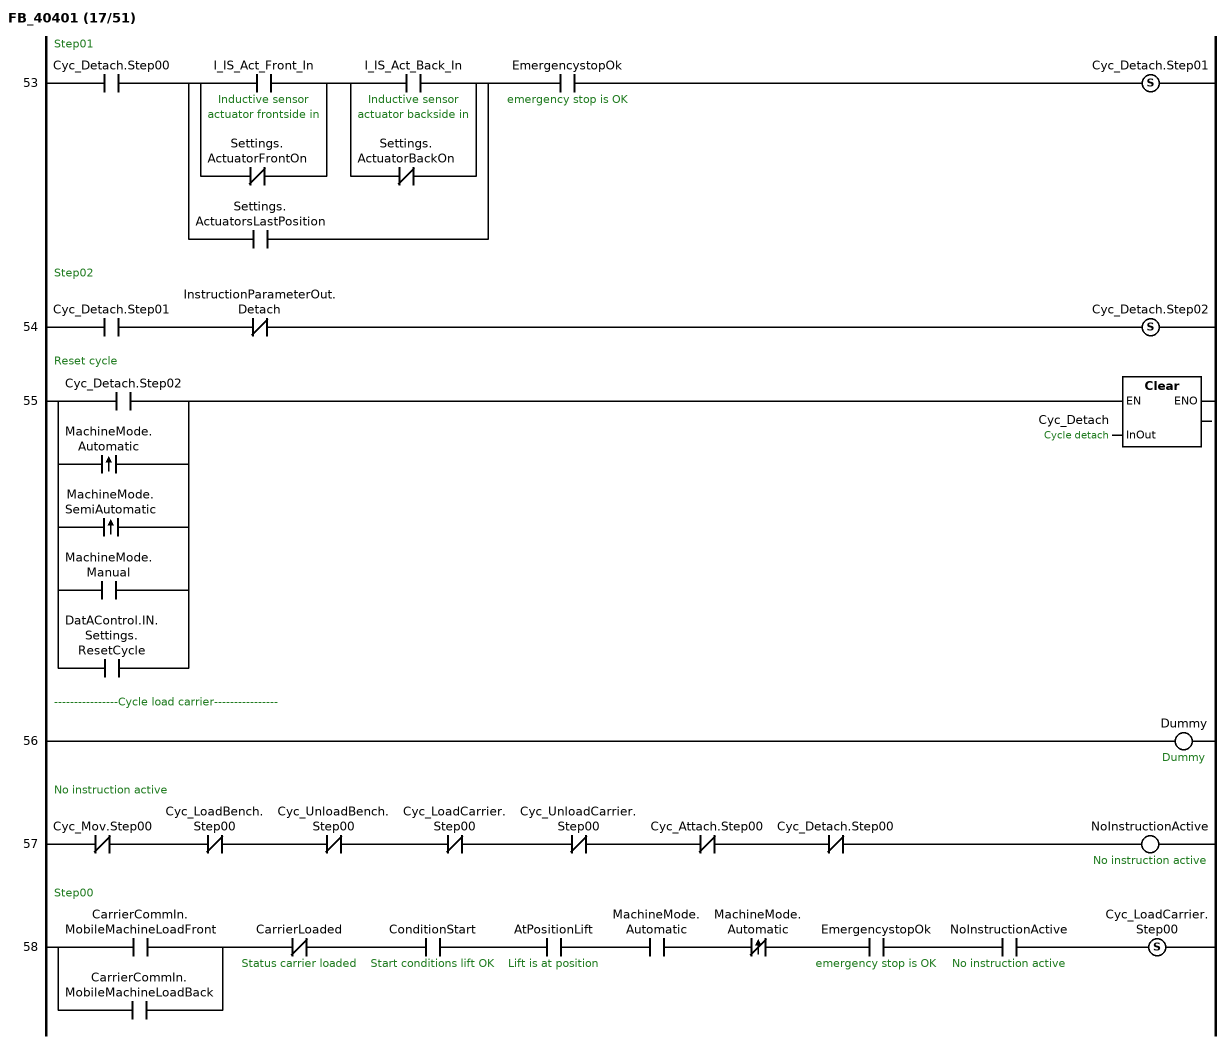
(* [picture p150: FB_40401, rungs 53-58] *)
(* Rung 53: Step01 *)
IF Cyc_Detach.Step00 AND (((I_IS_Act_Front_In OR NOT Settings.ActuatorFrontOn) AND (I_IS_Act_Back_In OR NOT Settings.ActuatorBackOn)) OR Settings.ActuatorsLastPosition) AND EmergencystopOk THEN
    Cyc_Detach.Step01 := TRUE;
END_IF;
(* Rung 54: Step02 *)
IF Cyc_Detach.Step01 AND NOT InstructionParameterOut.Detach THEN Cyc_Detach.Step02 := TRUE; END_IF;
(* Rung 55: Reset cycle *)
_e31(CLK := MachineMode.Automatic);
_e32(CLK := MachineMode.SemiAutomatic);
IF Cyc_Detach.Step02 OR _e31.Q OR _e32.Q OR MachineMode.Manual OR DatAControl.IN.Settings.ResetCycle THEN
    Clear(InOut := Cyc_Detach);
END_IF;
(* Rung 56: ----------------Cycle load carrier---------------- *)
Dummy := TRUE;
(* Rung 57: No instruction active *)
NoInstructionActive := NOT Cyc_Mov.Step00 AND NOT Cyc_LoadBench.Step00 AND NOT Cyc_UnloadBench.Step00 AND NOT Cyc_LoadCarrier.Step00 AND NOT Cyc_UnloadCarrier.Step00 AND NOT Cyc_Attach.Step00 AND NOT Cyc_Detach.Step00;
(* Rung 58: Step00 *)
_e33(CLK := MachineMode.Automatic);
IF (CarrierCommIn.MobileMachineLoadFront OR CarrierCommIn.MobileMachineLoadBack) AND NOT CarrierLoaded AND ConditionStart AND AtPositionLift AND MachineMode.Automatic AND NOT _e33.Q AND EmergencystopOk AND NoInstructionActive THEN
    Cyc_LoadCarrier.Step00 := TRUE;
END_IF;

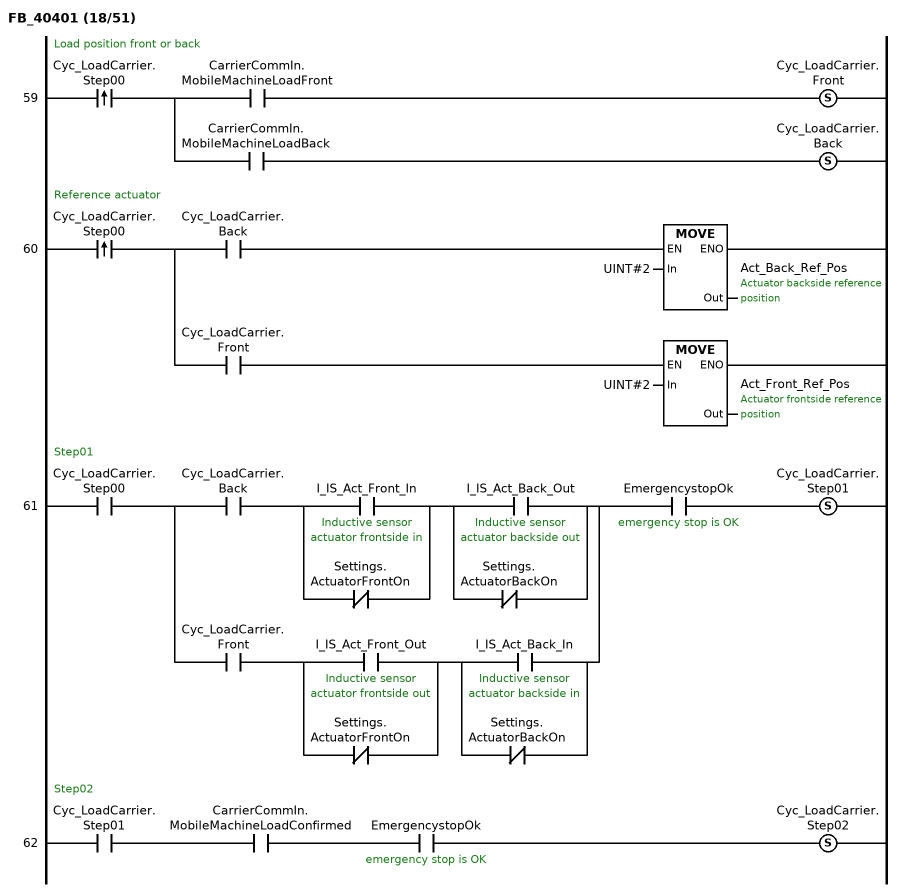
(* Rung 59: Load position front or back *)
_e34(CLK := Cyc_LoadCarrier.Step00);
IF _e34.Q AND CarrierCommIn.MobileMachineLoadFront THEN Cyc_LoadCarrier.Front := TRUE; END_IF;
IF _e34.Q AND CarrierCommIn.MobileMachineLoadBack THEN Cyc_LoadCarrier.Back := TRUE; END_IF;
(* Rung 60: Reference actuator *)
_e35(CLK := Cyc_LoadCarrier.Step00);
IF _e35.Q AND Cyc_LoadCarrier.Back THEN Act_Back_Ref_Pos := UINT#2; END_IF;
IF _e35.Q AND Cyc_LoadCarrier.Front THEN Act_Front_Ref_Pos := UINT#2; END_IF;
(* Rung 61: Step01 *)
IF Cyc_LoadCarrier.Step00 AND ((Cyc_LoadCarrier.Back AND (I_IS_Act_Front_In OR NOT Settings.ActuatorFrontOn) AND (I_IS_Act_Back_Out OR NOT Settings.ActuatorBackOn)) OR (Cyc_LoadCarrier.Front AND (I_IS_Act_Front_Out OR NOT Settings.ActuatorFrontOn) AND (I_IS_Act_Back_In OR NOT Settings.ActuatorBackOn))) AND EmergencystopOk THEN
    Cyc_LoadCarrier.Step01 := TRUE;
END_IF;
(* Rung 62: Step02 *)
IF Cyc_LoadCarrier.Step01 AND CarrierCommIn.MobileMachineLoadConfirmed AND EmergencystopOk THEN
    Cyc_LoadCarrier.Step02 := TRUE;
END_IF;

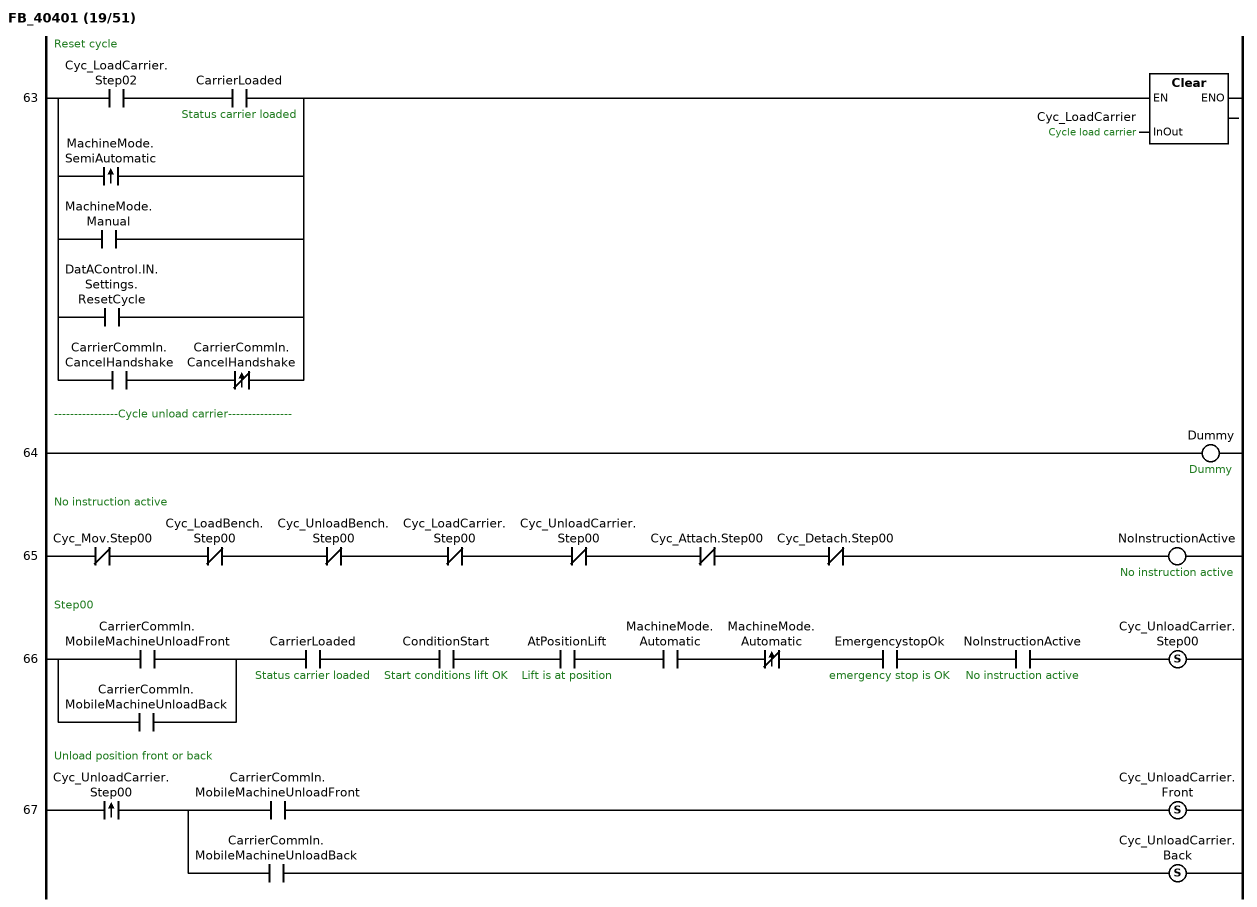
(* Rung 63: Reset cycle *)
_e36(CLK := MachineMode.SemiAutomatic);
_e37(CLK := CarrierCommIn.CancelHandshake);
IF (Cyc_LoadCarrier.Step02 AND CarrierLoaded) OR _e36.Q OR MachineMode.Manual OR DatAControl.IN.Settings.ResetCycle OR (CarrierCommIn.CancelHandshake AND NOT _e37.Q) THEN
    Clear(InOut := Cyc_LoadCarrier);
END_IF;
(* Rung 64: ----------------Cycle unload carrier---------------- *)
Dummy := TRUE;
(* Rung 65: No instruction active *)
NoInstructionActive := NOT Cyc_Mov.Step00 AND NOT Cyc_LoadBench.Step00 AND NOT Cyc_UnloadBench.Step00 AND NOT Cyc_LoadCarrier.Step00 AND NOT Cyc_UnloadCarrier.Step00 AND NOT Cyc_Attach.Step00 AND NOT Cyc_Detach.Step00;
(* Rung 66: Step00 *)
_e38(CLK := MachineMode.Automatic);
IF (CarrierCommIn.MobileMachineUnloadFront OR CarrierCommIn.MobileMachineUnloadBack) AND CarrierLoaded AND ConditionStart AND AtPositionLift AND MachineMode.Automatic AND NOT _e38.Q AND EmergencystopOk AND NoInstructionActive THEN
    Cyc_UnloadCarrier.Step00 := TRUE;
END_IF;
(* Rung 67: Unload position front or back *)
_e39(CLK := Cyc_UnloadCarrier.Step00);
IF _e39.Q AND CarrierCommIn.MobileMachineUnloadFront THEN Cyc_UnloadCarrier.Front := TRUE; END_IF;
IF _e39.Q AND CarrierCommIn.MobileMachineUnloadBack THEN Cyc_UnloadCarrier.Back := TRUE; END_IF;

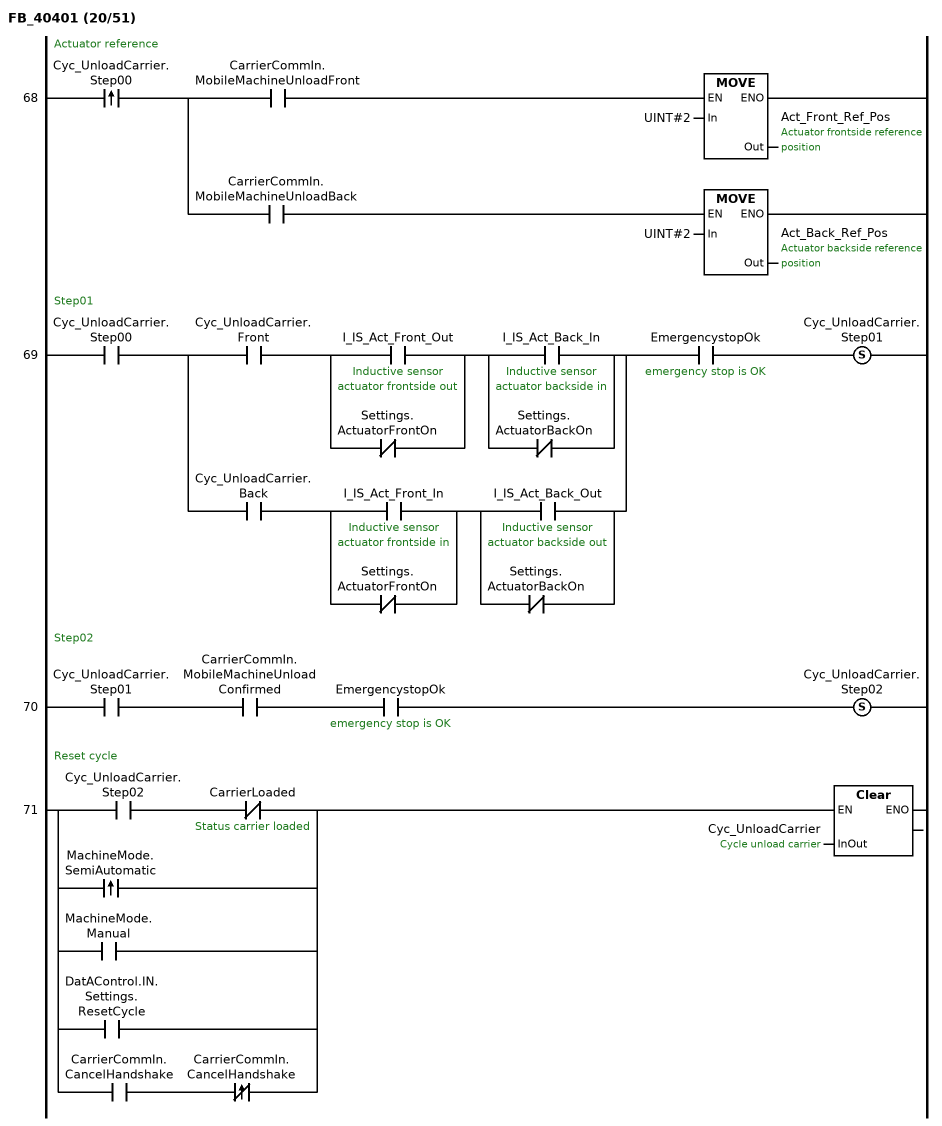
(* Rung 68: Actuator reference *)
_e40(CLK := Cyc_UnloadCarrier.Step00);
IF _e40.Q AND CarrierCommIn.MobileMachineUnloadFront THEN Act_Front_Ref_Pos := UINT#2; END_IF;
IF _e40.Q AND CarrierCommIn.MobileMachineUnloadBack THEN Act_Back_Ref_Pos := UINT#2; END_IF;
(* Rung 69: Step01 *)
IF Cyc_UnloadCarrier.Step00 AND ((Cyc_UnloadCarrier.Front AND (I_IS_Act_Front_Out OR NOT Settings.ActuatorFrontOn) AND (I_IS_Act_Back_In OR NOT Settings.ActuatorBackOn)) OR (Cyc_UnloadCarrier.Back AND (I_IS_Act_Front_In OR NOT Settings.ActuatorFrontOn) AND (I_IS_Act_Back_Out OR NOT Settings.ActuatorBackOn))) AND EmergencystopOk THEN
    Cyc_UnloadCarrier.Step01 := TRUE;
END_IF;
(* Rung 70: Step02 *)
IF Cyc_UnloadCarrier.Step01 AND CarrierCommIn.MobileMachineUnloadConfirmed AND EmergencystopOk THEN
    Cyc_UnloadCarrier.Step02 := TRUE;
END_IF;
(* Rung 71: Reset cycle *)
_e41(CLK := MachineMode.SemiAutomatic);
_e42(CLK := CarrierCommIn.CancelHandshake);
IF (Cyc_UnloadCarrier.Step02 AND NOT CarrierLoaded) OR _e41.Q OR MachineMode.Manual OR DatAControl.IN.Settings.ResetCycle OR (CarrierCommIn.CancelHandshake AND NOT _e42.Q) THEN
    Clear(InOut := Cyc_UnloadCarrier);
END_IF;

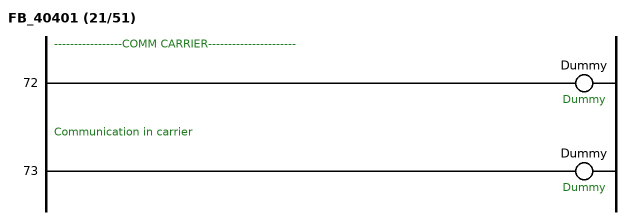
(* Rung 72: -----------------COMM CARRIER---------------------- *)
Dummy := TRUE;
(* Rung 73: Communication in carrier *)
Dummy := TRUE;

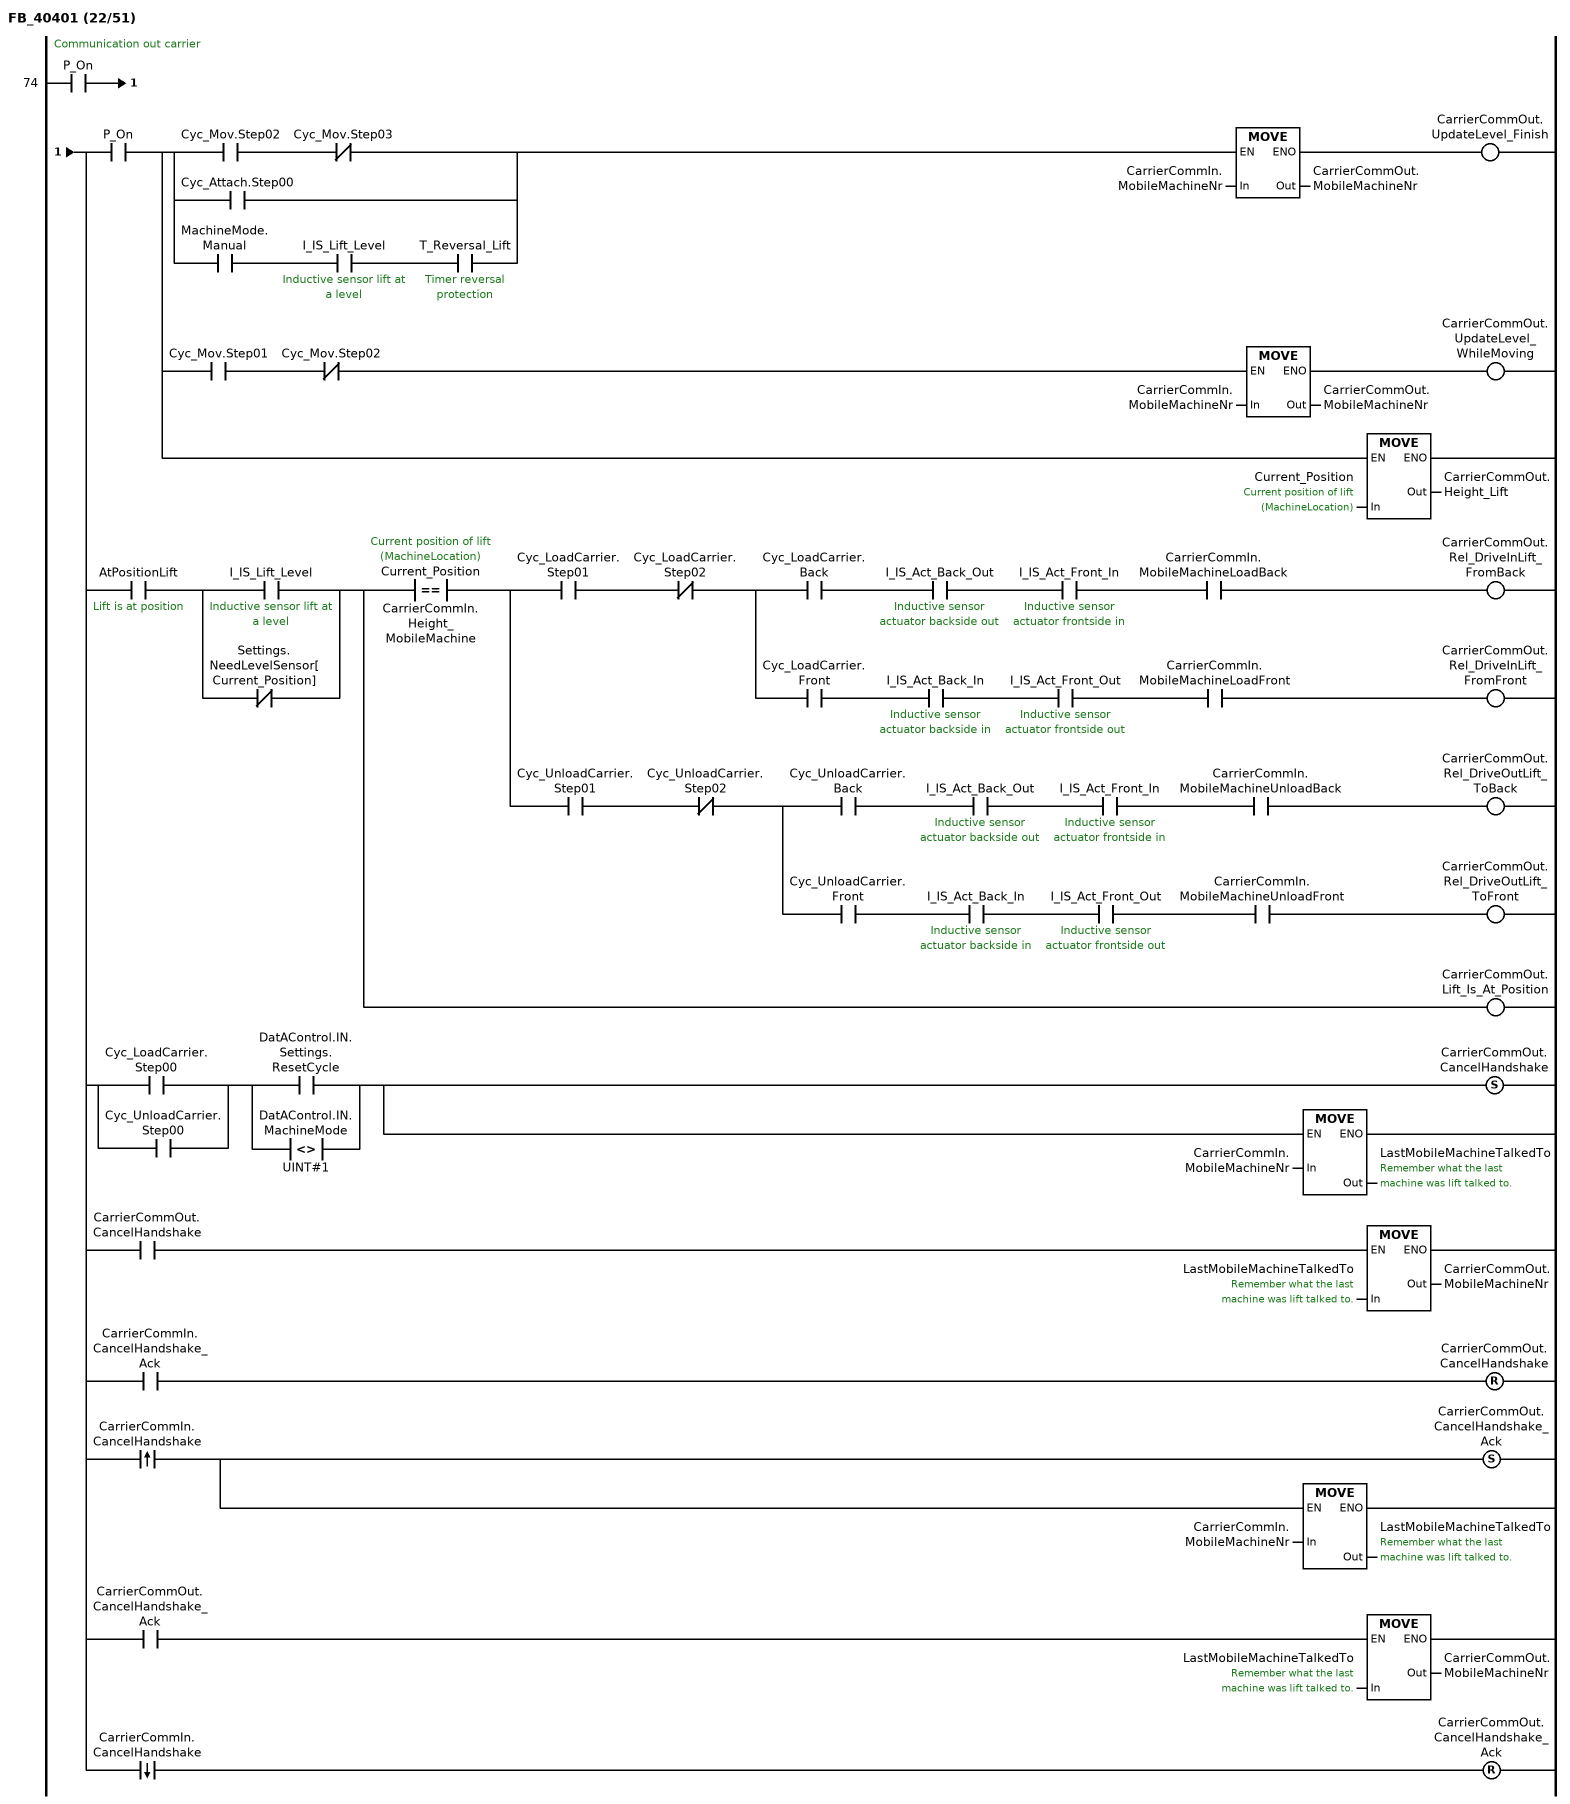
(* Rung 74: Communication out carrier *)
IF P_On AND P_On AND ((Cyc_Mov.Step02 AND NOT Cyc_Mov.Step03) OR Cyc_Attach.Step00 OR (MachineMode.Manual AND I_IS_Lift_Level AND T_Reversal_Lift)) THEN
    CarrierCommOut.MobileMachineNr := CarrierCommIn.MobileMachineNr;
END_IF;
CarrierCommOut.UpdateLevel_Finish := P_On AND P_On AND ((Cyc_Mov.Step02 AND NOT Cyc_Mov.Step03) OR Cyc_Attach.Step00 OR (MachineMode.Manual AND I_IS_Lift_Level AND T_Reversal_Lift));
IF P_On AND P_On AND Cyc_Mov.Step01 AND NOT Cyc_Mov.Step02 THEN
    CarrierCommOut.MobileMachineNr := CarrierCommIn.MobileMachineNr;
END_IF;
CarrierCommOut.UpdateLevel_WhileMoving := P_On AND P_On AND Cyc_Mov.Step01 AND NOT Cyc_Mov.Step02;
IF P_On AND P_On THEN CarrierCommOut.Height_Lift := Current_Position; END_IF;
_p43 := P_On AND AtPositionLift AND (I_IS_Lift_Level OR NOT Settings.NeedLevelSensor[Current_Position]);
_p44 := _p43 AND (Current_Position = CarrierCommIn.Height_MobileMachine);
_p45 := _p44 AND Cyc_LoadCarrier.Step01 AND NOT Cyc_LoadCarrier.Step02;
CarrierCommOut.Rel_DriveInLift_FromBack := _p45 AND Cyc_LoadCarrier.Back AND I_IS_Act_Back_Out AND I_IS_Act_Front_In AND CarrierCommIn.MobileMachineLoadBack;
CarrierCommOut.Rel_DriveInLift_FromFront := _p45 AND Cyc_LoadCarrier.Front AND I_IS_Act_Back_In AND I_IS_Act_Front_Out AND CarrierCommIn.MobileMachineLoadFront;
_p46 := _p44 AND Cyc_UnloadCarrier.Step01 AND NOT Cyc_UnloadCarrier.Step02;
CarrierCommOut.Rel_DriveOutLift_ToBack := _p46 AND Cyc_UnloadCarrier.Back AND I_IS_Act_Back_Out AND I_IS_Act_Front_In AND CarrierCommIn.MobileMachineUnloadBack;
CarrierCommOut.Rel_DriveOutLift_ToFront := _p46 AND Cyc_UnloadCarrier.Front AND I_IS_Act_Back_In AND I_IS_Act_Front_Out AND CarrierCommIn.MobileMachineUnloadFront;
CarrierCommOut.Lift_Is_At_Position := _p43;
_p47 := P_On AND (Cyc_LoadCarrier.Step00 OR Cyc_UnloadCarrier.Step00) AND (DatAControl.IN.Settings.ResetCycle OR (DatAControl.IN.MachineMode <> UINT#1));
IF _p47 THEN
    CarrierCommOut.CancelHandshake := TRUE;
    LastMobileMachineTalkedTo := CarrierCommIn.MobileMachineNr;
END_IF;
IF P_On AND CarrierCommOut.CancelHandshake THEN
    CarrierCommOut.MobileMachineNr := LastMobileMachineTalkedTo;
END_IF;
IF P_On AND CarrierCommIn.CancelHandshake_Ack THEN CarrierCommOut.CancelHandshake := FALSE; END_IF;
_e48(CLK := CarrierCommIn.CancelHandshake);
IF P_On AND _e48.Q THEN
    CarrierCommOut.CancelHandshake_Ack := TRUE;
    LastMobileMachineTalkedTo := CarrierCommIn.MobileMachineNr;
END_IF;
IF P_On AND CarrierCommOut.CancelHandshake_Ack THEN
    CarrierCommOut.MobileMachineNr := LastMobileMachineTalkedTo;
END_IF;
_e49(CLK := CarrierCommIn.CancelHandshake);
IF P_On AND _e49.Q THEN CarrierCommOut.CancelHandshake_Ack := FALSE; END_IF;

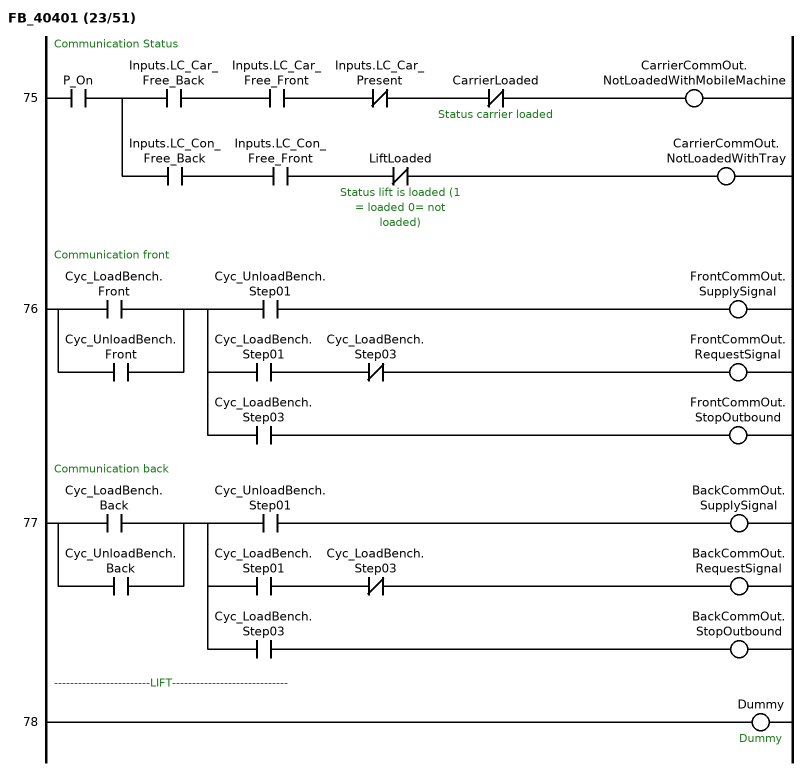
(* Rung 75: Communication Status *)
CarrierCommOut.NotLoadedWithMobileMachine := P_On AND Inputs.LC_Car_Free_Back AND Inputs.LC_Car_Free_Front AND NOT Inputs.LC_Car_Present AND NOT CarrierLoaded;
CarrierCommOut.NotLoadedWithTray := P_On AND Inputs.LC_Con_Free_Back AND Inputs.LC_Con_Free_Front AND NOT LiftLoaded;
(* Rung 76: Communication front *)
FrontCommOut.SupplySignal := (Cyc_LoadBench.Front OR Cyc_UnloadBench.Front) AND Cyc_UnloadBench.Step01;
FrontCommOut.RequestSignal := (Cyc_LoadBench.Front OR Cyc_UnloadBench.Front) AND Cyc_LoadBench.Step01 AND NOT Cyc_LoadBench.Step03;
FrontCommOut.StopOutbound := (Cyc_LoadBench.Front OR Cyc_UnloadBench.Front) AND Cyc_LoadBench.Step03;
(* Rung 77: Communication back *)
BackCommOut.SupplySignal := (Cyc_LoadBench.Back OR Cyc_UnloadBench.Back) AND Cyc_UnloadBench.Step01;
BackCommOut.RequestSignal := (Cyc_LoadBench.Back OR Cyc_UnloadBench.Back) AND Cyc_LoadBench.Step01 AND NOT Cyc_LoadBench.Step03;
BackCommOut.StopOutbound := (Cyc_LoadBench.Back OR Cyc_UnloadBench.Back) AND Cyc_LoadBench.Step03;
(* Rung 78: ------------------------LIFT----------------------------- *)
Dummy := TRUE;

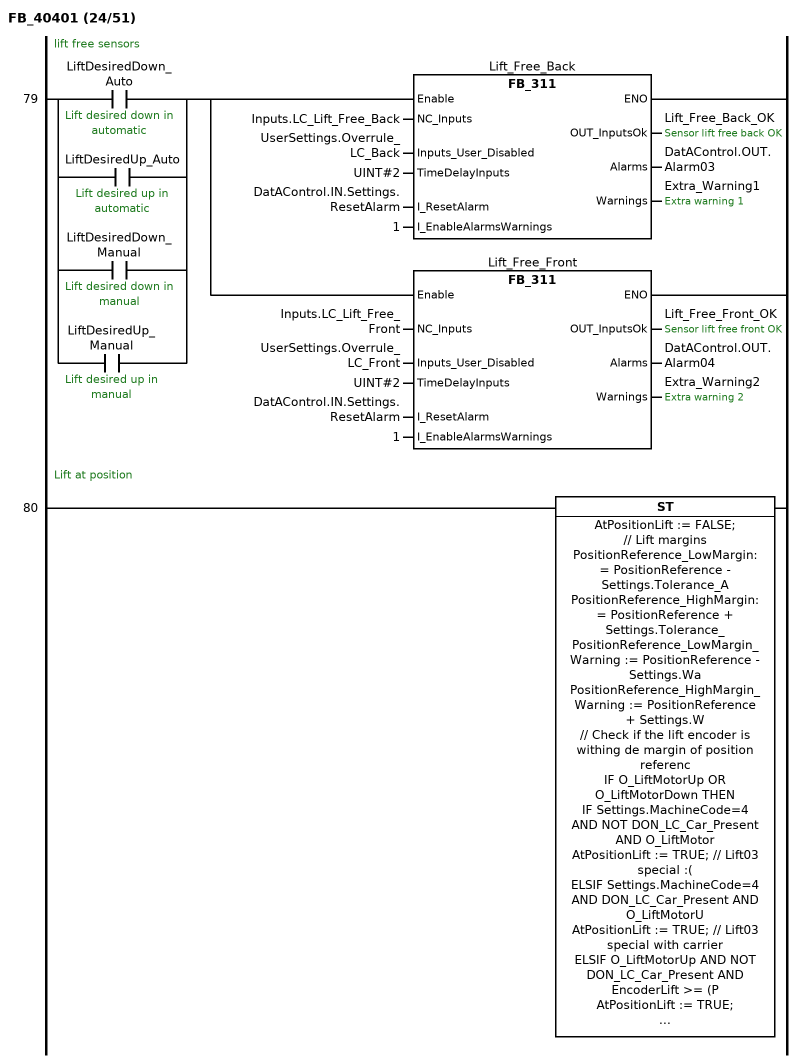
(* Rung 79: lift free sensors *)
_p50 := LiftDesiredDown_Auto OR LiftDesiredUp_Auto OR LiftDesiredDown_Manual OR LiftDesiredUp_Manual;
Lift_Free_Back(Enable := _p50, NC_Inputs := Inputs.LC_Lift_Free_Back, Inputs_User_Disabled := UserSettings.Overrule_LC_Back, TimeDelayInputs := UINT#2, I_ResetAlarm := DatAControl.IN.Settings.ResetAlarm, I_EnableAlarmsWarnings := 1, OUT_InputsOk => Lift_Free_Back_OK, Alarms => DatAControl.OUT.Alarm03, Warnings => Extra_Warning1);
Lift_Free_Front(Enable := _p50, NC_Inputs := Inputs.LC_Lift_Free_Front, Inputs_User_Disabled := UserSettings.Overrule_LC_Front, TimeDelayInputs := UINT#2, I_ResetAlarm := DatAControl.IN.Settings.ResetAlarm, I_EnableAlarmsWarnings := 1, OUT_InputsOk => Lift_Free_Front_OK, Alarms => DatAControl.OUT.Alarm04, Warnings => Extra_Warning2);
(* Rung 80: Lift at position *)
AtPositionLift := FALSE;

// Lift margins
PositionReference_LowMargin:= PositionReference - Settings.Tolerance_At_Position;
PositionReference_HighMargin:= PositionReference + Settings.Tolerance_At_Position;
PositionReference_LowMargin_Warning := PositionReference - Settings.Warning_Tolerance_At_Position;
PositionReference_HighMargin_Warning := PositionReference + Settings.Warning_Tolerance_At_Position;

// Check if the lift encoder is withing de margin of position reference
IF O_LiftMotorUp OR O_LiftMotorDown THEN
	IF Settings.MachineCode=4 AND NOT DON_LC_Car_Present AND O_LiftMotorUp AND EncoderLift >= (PositionReference + 25) AND EncoderLift <= (PositionReference_HighMargin) THEN // EncoderLiftOvershootUp
		AtPositionLift := TRUE; // Lift03 special :(
	ELSIF Settings.MachineCode=4 AND DON_LC_Car_Present AND O_LiftMotorUp AND EncoderLift >= (PositionReference + 25) AND EncoderLift <= (PositionReference_HighMargin) THEN
		AtPositionLift := TRUE; // Lift03 special with carrier
	ELSIF O_LiftMotorUp AND NOT DON_LC_Car_Present AND EncoderLift >= (PositionReference - EncoderLiftOvershootUp) AND EncoderLift <= PositionReference_HighMargin THEN
		AtPositionLift := TRUE;
	ELSIF O_LiftMotorUp AND DON_LC_Car_Present AND EncoderLift >= (PositionReference - EncoderLiftOvershootUp - EncoderLiftOvershootUp) AND EncoderLift <= PositionReference_HighMargin THEN
		AtPositionLift := TRUE; // with carrier
	ELSIF Settings.MachineCode=4 AND O_LiftMotorDown AND NOT DON_LC_Car_Present AND EncoderLift <= (PositionReference + 45) AND EncoderLift >= PositionReference_LowMargin  THEN
		AtPositionLift := TRUE; // Lift03 special :)
	ELSIF Settings.MachineCode=4 AND O_LiftMotorDown AND DON_LC_Car_Present AND EncoderLift <= (PositionReference + 45) AND EncoderLift >= PositionReference_LowMargin  THEN
		AtPositionLift := TRUE; // Lift03 special with carrier
	ELSIF O_LiftMotorDown AND NOT DON_LC_Car_Present AND EncoderLift <= (PositionReference + EncoderLiftOvershootDown) AND EncoderLift >= PositionReference_LowMargin THEN
		AtPositionLift := TRUE;
	ELSIF O_LiftMotorDown AND DON_LC_Car_Present AND EncoderLift <= (PositionReference + EncoderLiftOvershootDown + EncoderLiftOvershootDown) AND EncoderLift >= PositionReference_LowMargin THEN
		AtPositionLift := TRUE; // with carrier
	END_IF;
ELSE
	IF (EncoderLift >= PositionReference_LowMargin) AND (EncoderLift <= PositionReference_HighMargin) THEN
		AtPositionLift := TRUE;
	END_IF;
END_IF;

Warning_AtPositionLift := FALSE;
IF AtPositionLift AND T_Reversal_Lift AND ((EncoderLift <= PositionReference_LowMargin_Warning) OR (EncoderLift >= PositionReference_HighMargin_Warning)) THEN
	Warning_AtPositionLift := TRUE;
END_IF;

Extra_Warning3 := WORD#0;

IF Warning_AtPositionLift THEN
	OutABit(Extra_Warning3,0,TRUE);
END_IF;

// Check for each position if the lift encoder is within the margins
FOR index:=1 TO 16 BY 1 DO
	IF (EncoderLift >= ( Settings.PulseLevel[index] - Settings.Tolerance_At_Position)) AND (EncoderLift <= (Settings.PulseLevel[index] + Settings.Tolerance_At_Position)) THEN
		Current_Position:= index;
	END_IF;
END_FOR;

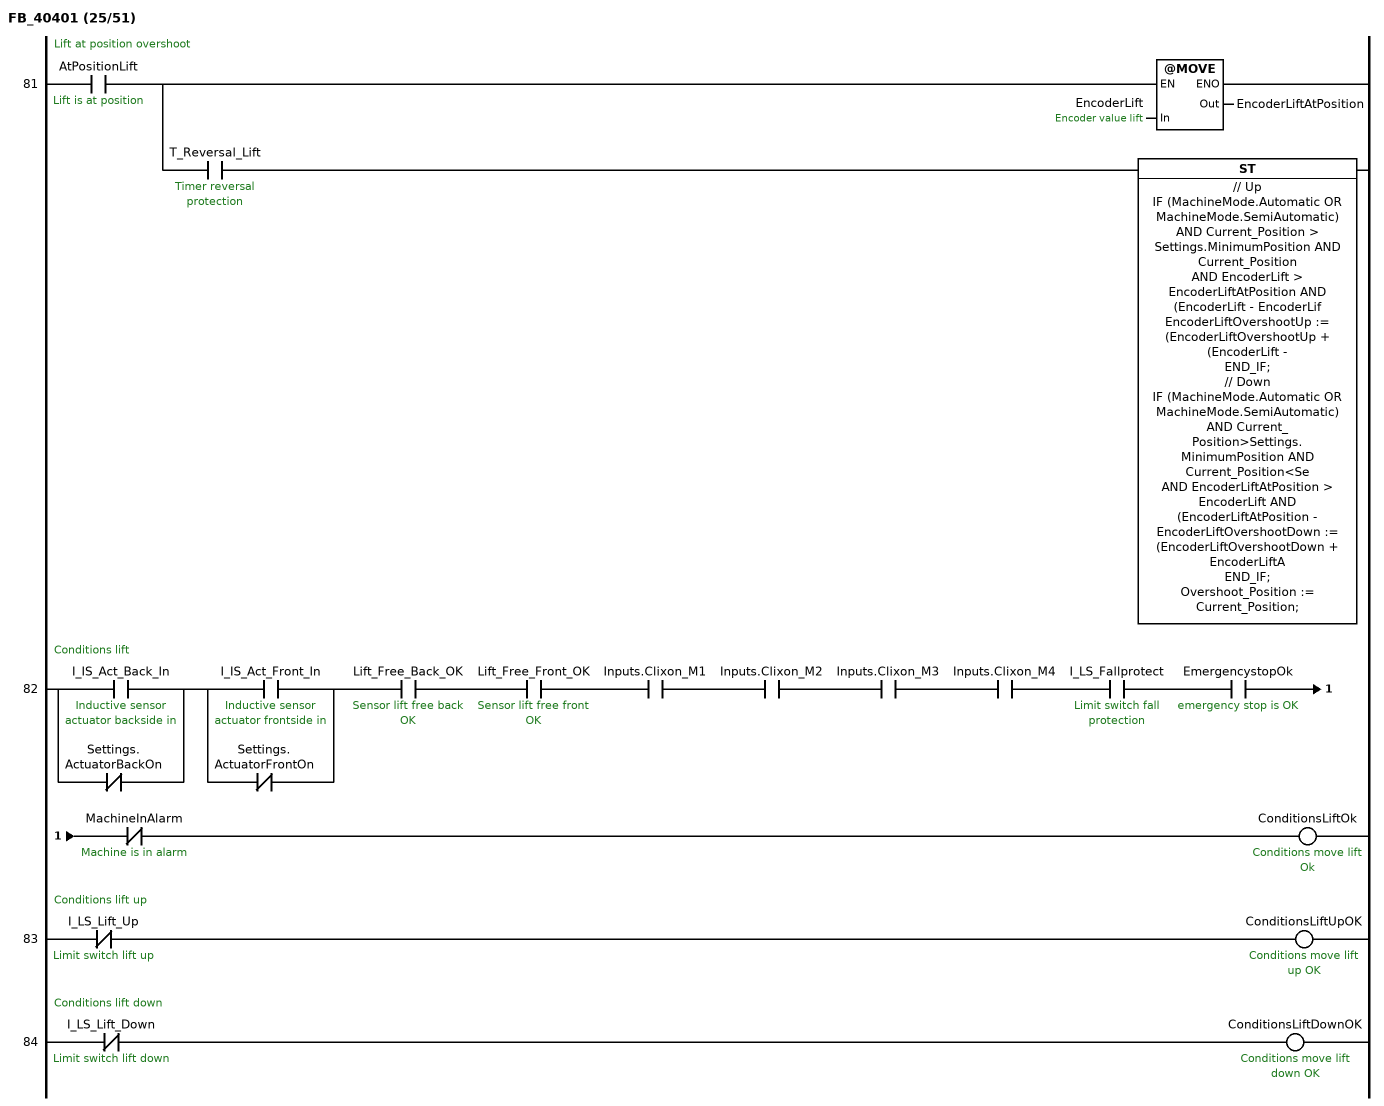
(* Rung 81: Lift at position overshoot *)
_e51(CLK := AtPositionLift);
IF _e51.Q THEN EncoderLiftAtPosition := EncoderLift; END_IF;
IF AtPositionLift AND T_Reversal_Lift THEN
    // Up
    IF (MachineMode.Automatic OR MachineMode.SemiAutomatic)
     AND Current_Position > Settings.MinimumPosition AND Current_Position < Settings.MaximumPosition AND Current_Position <> Overshoot_Position
     AND EncoderLift > EncoderLiftAtPosition AND (EncoderLift - EncoderLiftAtPosition) < (Settings.Tolerance_At_Position*2) THEN
    		EncoderLiftOvershootUp := (EncoderLiftOvershootUp + (EncoderLift - EncoderLiftAtPosition))/2;
    END_IF;
    // Down
    IF (MachineMode.Automatic OR MachineMode.SemiAutomatic)
     AND Current_Position>Settings.MinimumPosition AND Current_Position<Settings.MaximumPosition AND Current_Position<>Overshoot_Position
     AND EncoderLiftAtPosition > EncoderLift AND (EncoderLiftAtPosition - EncoderLift) < (Settings.Tolerance_At_Position*2) THEN
    	EncoderLiftOvershootDown := (EncoderLiftOvershootDown + EncoderLiftAtPosition - EncoderLift)/2;
    END_IF;
    
    Overshoot_Position := Current_Position;
END_IF;
(* Rung 82: Conditions lift *)
ConditionsLiftOk := (I_IS_Act_Back_In OR NOT Settings.ActuatorBackOn) AND (I_IS_Act_Front_In OR NOT Settings.ActuatorFrontOn) AND Lift_Free_Back_OK AND Lift_Free_Front_OK AND Inputs.Clixon_M1 AND Inputs.Clixon_M2 AND Inputs.Clixon_M3 AND Inputs.Clixon_M4 AND I_LS_Fallprotect AND EmergencystopOk AND NOT MachineInAlarm;
(* Rung 83: Conditions lift up *)
ConditionsLiftUpOK := NOT I_LS_Lift_Up;
(* Rung 84: Conditions lift down *)
ConditionsLiftDownOK := NOT I_LS_Lift_Down;

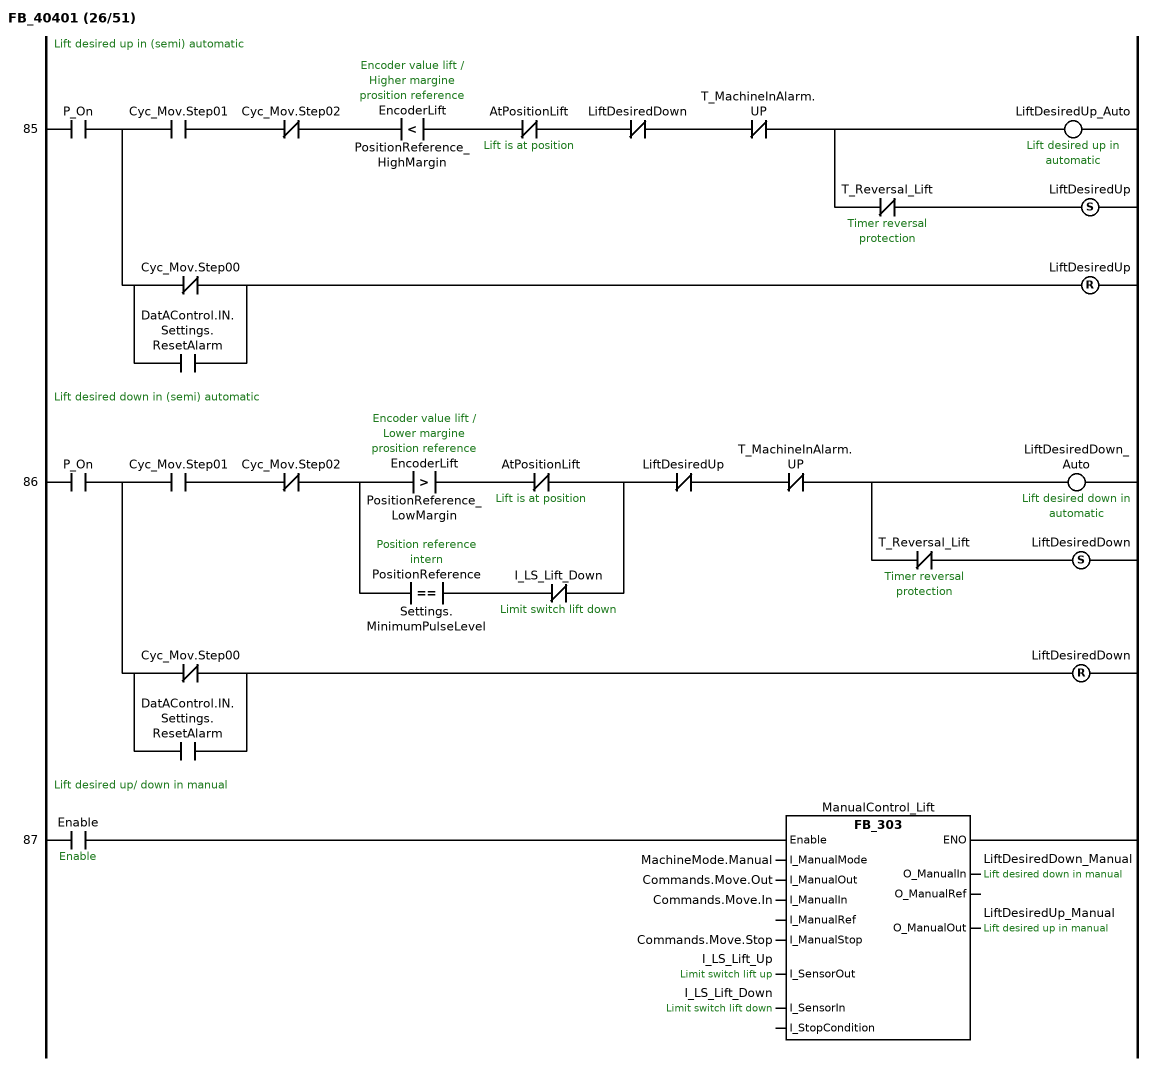
(* Rung 85: Lift desired up in (semi) automatic *)
_p52 := P_On AND Cyc_Mov.Step01 AND NOT Cyc_Mov.Step02 AND (EncoderLift < PositionReference_HighMargin) AND NOT AtPositionLift AND NOT LiftDesiredDown AND NOT T_MachineInAlarm.UP;
LiftDesiredUp_Auto := _p52;
IF _p52 AND NOT T_Reversal_Lift THEN LiftDesiredUp := TRUE; END_IF;
IF P_On AND (NOT Cyc_Mov.Step00 OR DatAControl.IN.Settings.ResetAlarm) THEN
    LiftDesiredUp := FALSE;
END_IF;
(* Rung 86: Lift desired down in (semi) automatic *)
_p53 := P_On AND Cyc_Mov.Step01 AND NOT Cyc_Mov.Step02 AND (((EncoderLift > PositionReference_LowMargin) AND NOT AtPositionLift) OR ((PositionReference = Settings.MinimumPulseLevel) AND NOT I_LS_Lift_Down)) AND NOT LiftDesiredUp AND NOT T_MachineInAlarm.UP;
LiftDesiredDown_Auto := _p53;
IF _p53 AND NOT T_Reversal_Lift THEN LiftDesiredDown := TRUE; END_IF;
IF P_On AND (NOT Cyc_Mov.Step00 OR DatAControl.IN.Settings.ResetAlarm) THEN
    LiftDesiredDown := FALSE;
END_IF;
(* Rung 87: Lift desired up/ down in manual *)
ManualControl_Lift(Enable := Enable, I_ManualMode := MachineMode.Manual, I_ManualOut := Commands.Move.Out, I_ManualIn := Commands.Move.In, I_ManualStop := Commands.Move.Stop, I_SensorOut := I_LS_Lift_Up, I_SensorIn := I_LS_Lift_Down, O_ManualIn => LiftDesiredDown_Manual, O_ManualOut => LiftDesiredUp_Manual);

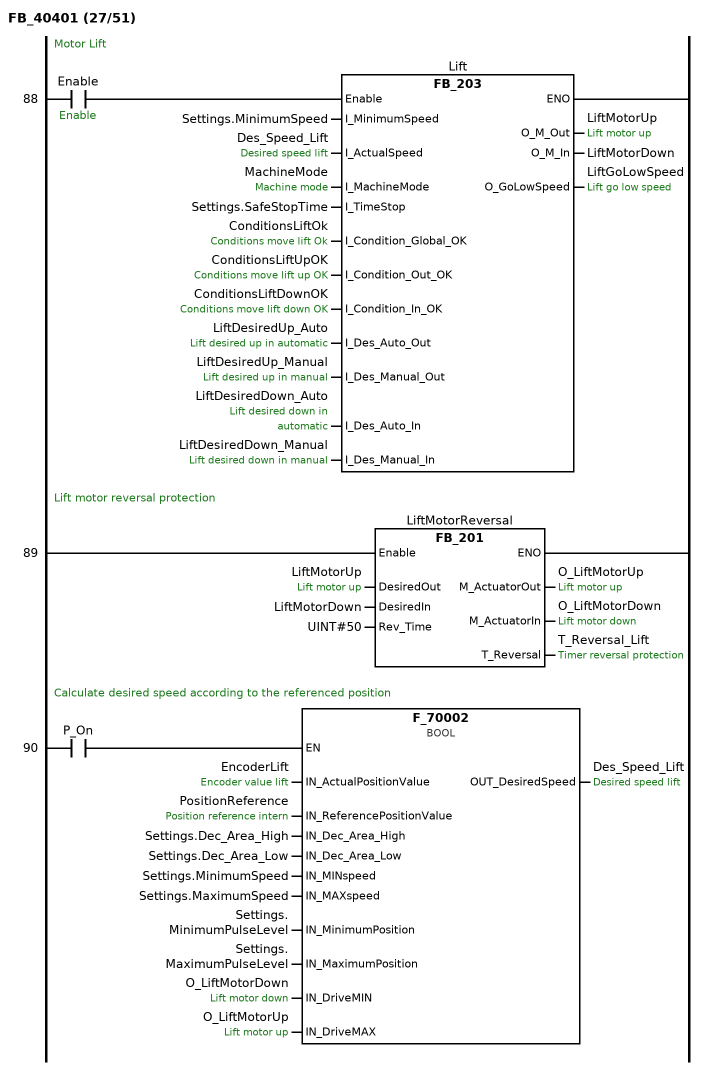
(* Rung 88: Motor Lift *)
Lift(Enable := Enable, I_MinimumSpeed := Settings.MinimumSpeed, I_ActualSpeed := Des_Speed_Lift, I_MachineMode := MachineMode, I_TimeStop := Settings.SafeStopTime, I_Condition_Global_OK := ConditionsLiftOk, I_Condition_Out_OK := ConditionsLiftUpOK, I_Condition_In_OK := ConditionsLiftDownOK, I_Des_Auto_Out := LiftDesiredUp_Auto, I_Des_Manual_Out := LiftDesiredUp_Manual, I_Des_Auto_In := LiftDesiredDown_Auto, I_Des_Manual_In := LiftDesiredDown_Manual, O_M_Out => LiftMotorUp, O_M_In => LiftMotorDown, O_GoLowSpeed => LiftGoLowSpeed);
(* Rung 89: Lift motor reversal protection *)
LiftMotorReversal(Enable := TRUE, DesiredOut := LiftMotorUp, DesiredIn := LiftMotorDown, Rev_Time := UINT#50, M_ActuatorOut => O_LiftMotorUp, M_ActuatorIn => O_LiftMotorDown, T_Reversal => T_Reversal_Lift);
(* Rung 90: Calculate desired speed according to the referenced position *)
_t54 := FALSE;
IF P_On THEN _t54 := F_70002(IN_ActualPositionValue := EncoderLift, IN_ReferencePositionValue := PositionReference, IN_Dec_Area_High := Settings.Dec_Area_High, IN_Dec_Area_Low := Settings.Dec_Area_Low, IN_MINspeed := Settings.MinimumSpeed, IN_MAXspeed := Settings.MaximumSpeed, IN_MinimumPosition := Settings.MinimumPulseLevel, IN_MaximumPosition := Settings.MaximumPulseLevel, IN_DriveMIN := O_LiftMotorDown, IN_DriveMAX := O_LiftMotorUp, OUT_DesiredSpeed => Des_Speed_Lift); END_IF;

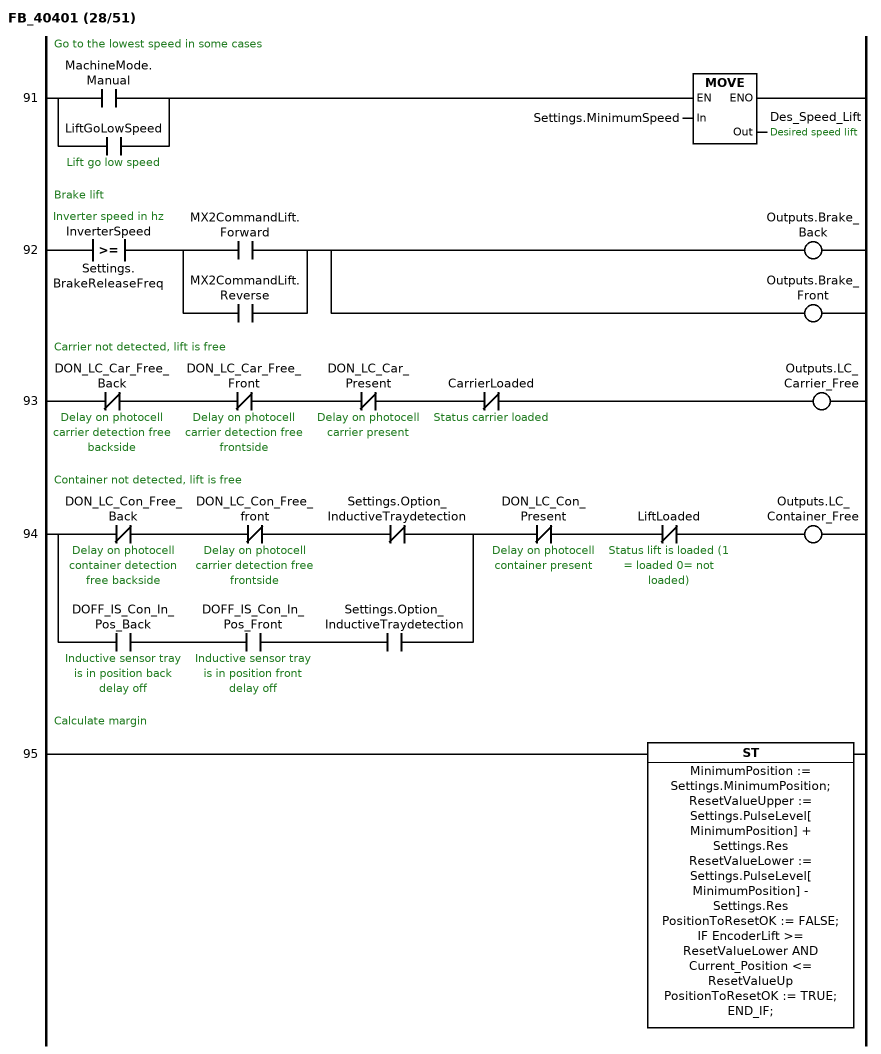
(* Rung 91: Go to the lowest speed in some cases *)
IF MachineMode.Manual OR LiftGoLowSpeed THEN Des_Speed_Lift := Settings.MinimumSpeed; END_IF;
(* Rung 92: Brake lift *)
_p55 := (InverterSpeed >= Settings.BrakeReleaseFreq) AND (MX2CommandLift.Forward OR MX2CommandLift.Reverse);
Outputs.Brake_Back := _p55;
Outputs.Brake_Front := _p55;
(* Rung 93: Carrier not detected, lift is free *)
Outputs.LC_Carrier_Free := NOT DON_LC_Car_Free_Back AND NOT DON_LC_Car_Free_Front AND NOT DON_LC_Car_Present AND NOT CarrierLoaded;
(* Rung 94: Container not detected, lift is free *)
Outputs.LC_Container_Free := ((NOT DON_LC_Con_Free_Back AND NOT DON_LC_Con_Free_front AND NOT Settings.Option_InductiveTraydetection) OR (DOFF_IS_Con_In_Pos_Back AND DOFF_IS_Con_In_Pos_Front AND Settings.Option_InductiveTraydetection)) AND NOT DON_LC_Con_Present AND NOT LiftLoaded;
(* Rung 95: Calculate margin *)
MinimumPosition := Settings.MinimumPosition;

ResetValueUpper := Settings.PulseLevel[MinimumPosition] + Settings.ResetValueMargin;
ResetValueLower := Settings.PulseLevel[MinimumPosition] - Settings.ResetValueMargin;

PositionToResetOK := FALSE;
IF EncoderLift >= ResetValueLower AND Current_Position <= ResetValueUpper THEN
	PositionToResetOK := TRUE;
END_IF;

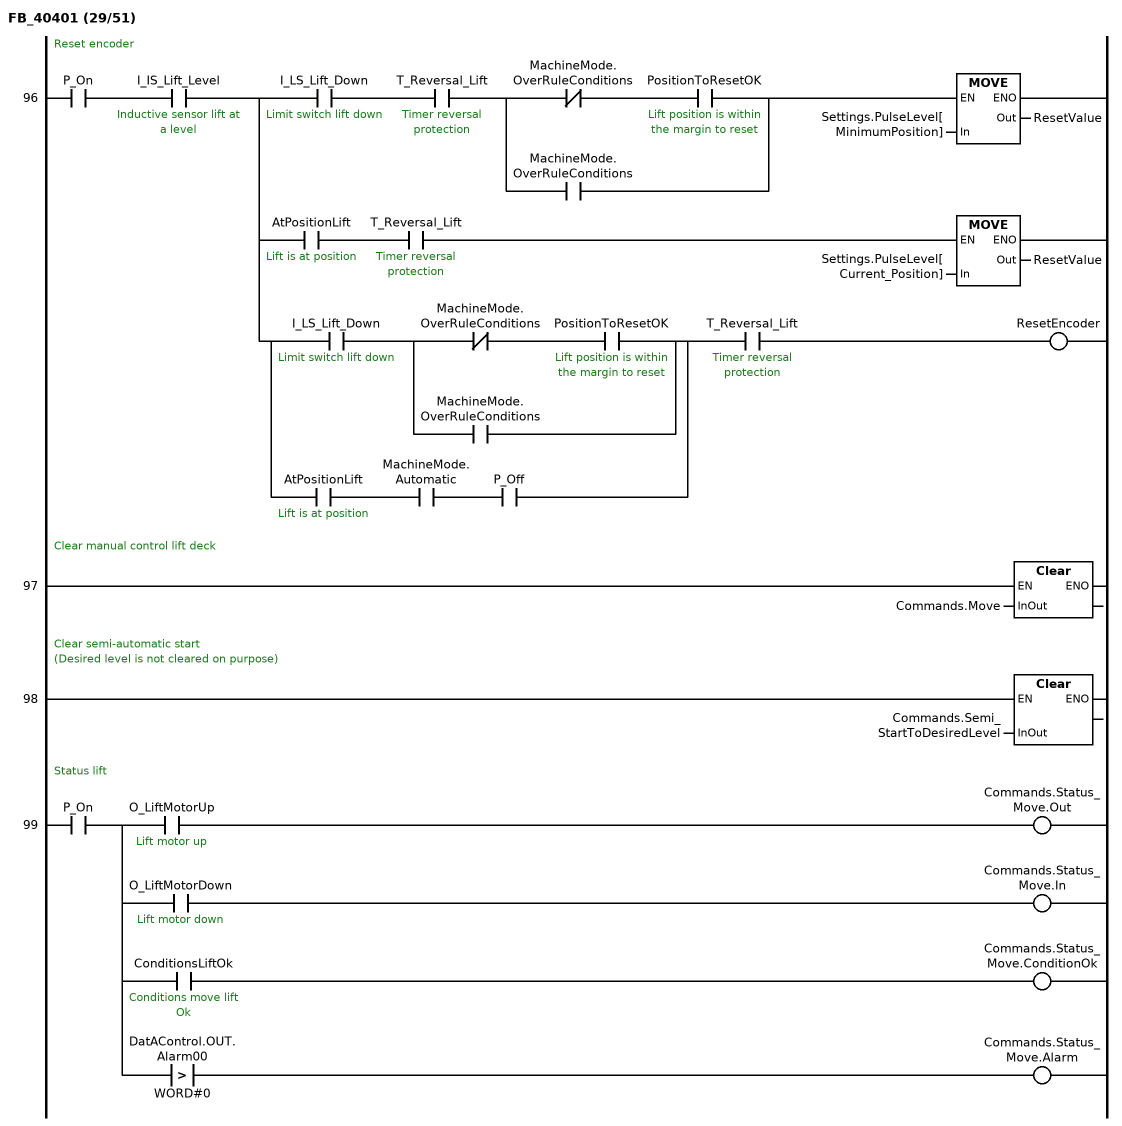
(* Rung 96: Reset encoder *)
IF P_On AND I_IS_Lift_Level AND I_LS_Lift_Down AND T_Reversal_Lift AND ((NOT MachineMode.OverRuleConditions AND PositionToResetOK) OR MachineMode.OverRuleConditions) THEN
    ResetValue := Settings.PulseLevel[MinimumPosition];
END_IF;
IF P_On AND I_IS_Lift_Level AND AtPositionLift AND T_Reversal_Lift THEN
    ResetValue := Settings.PulseLevel[Current_Position];
END_IF;
ResetEncoder := P_On AND I_IS_Lift_Level AND ((I_LS_Lift_Down AND ((NOT MachineMode.OverRuleConditions AND PositionToResetOK) OR MachineMode.OverRuleConditions)) OR (AtPositionLift AND MachineMode.Automatic AND P_Off)) AND T_Reversal_Lift;
(* Rung 97: Clear manual control lift deck *)
Clear(InOut := Commands.Move);
(* Rung 98: Clear semi-automatic start / (Desired level is not cleared on purpose) *)
Clear(InOut := Commands.Semi_StartToDesiredLevel);
(* Rung 99: Status lift *)
Commands.Status_Move.Out := P_On AND O_LiftMotorUp;
Commands.Status_Move.In := P_On AND O_LiftMotorDown;
Commands.Status_Move.ConditionOk := P_On AND ConditionsLiftOk;
Commands.Status_Move.Alarm := P_On AND (DatAControl.OUT.Alarm00 > WORD#0);

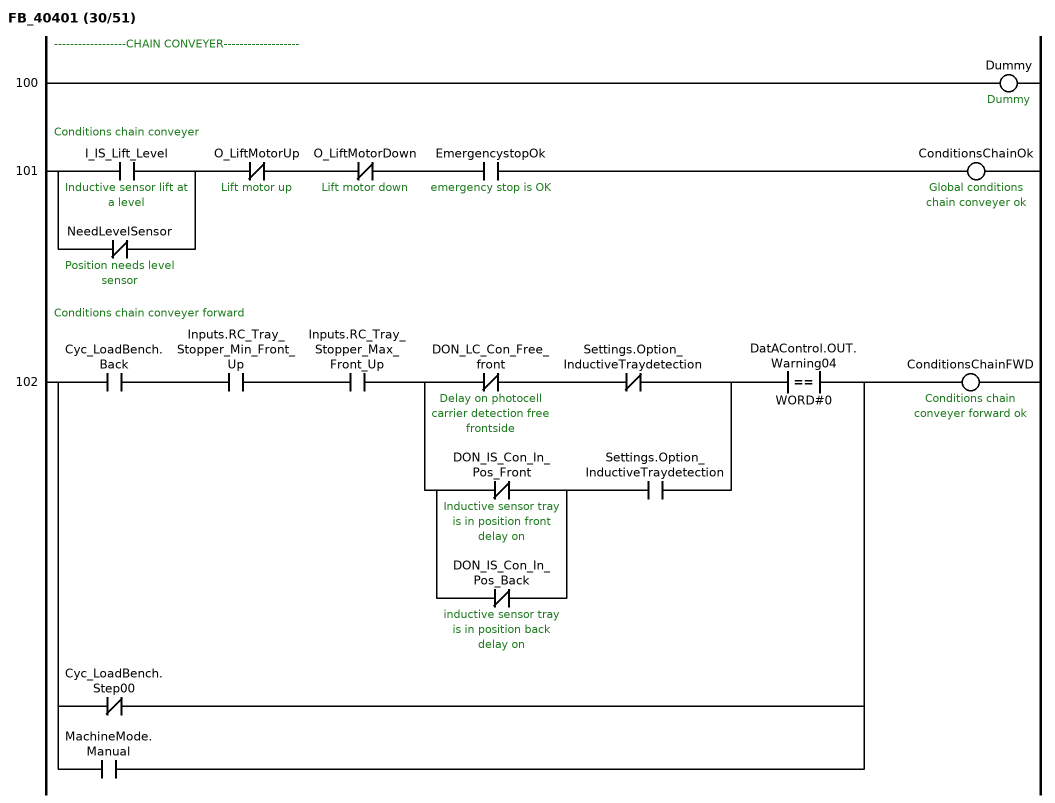
(* Rung 100: ------------------CHAIN CONVEYER------------------- *)
Dummy := TRUE;
(* Rung 101: Conditions chain conveyer *)
ConditionsChainOk := (I_IS_Lift_Level OR NOT NeedLevelSensor) AND NOT O_LiftMotorUp AND NOT O_LiftMotorDown AND EmergencystopOk;
(* Rung 102: Conditions chain conveyer forward *)
ConditionsChainFWD := (Cyc_LoadBench.Back AND Inputs.RC_Tray_Stopper_Min_Front_Up AND Inputs.RC_Tray_Stopper_Max_Front_Up AND ((NOT DON_LC_Con_Free_front AND NOT Settings.Option_InductiveTraydetection) OR ((NOT DON_IS_Con_In_Pos_Front OR NOT DON_IS_Con_In_Pos_Back) AND Settings.Option_InductiveTraydetection)) AND (DatAControl.OUT.Warning04 = WORD#0)) OR NOT Cyc_LoadBench.Step00 OR MachineMode.Manual;

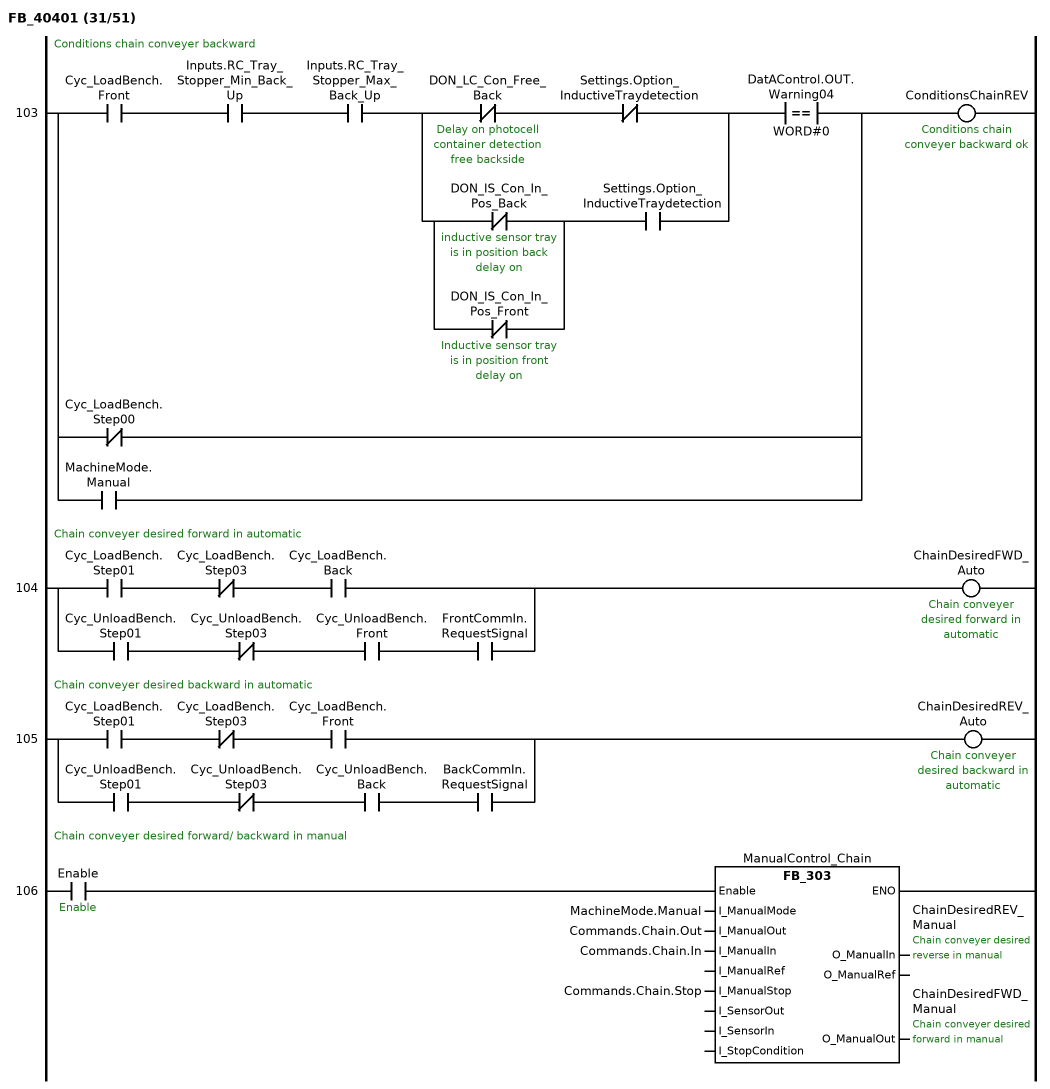
(* Rung 103: Conditions chain conveyer backward *)
ConditionsChainREV := (Cyc_LoadBench.Front AND Inputs.RC_Tray_Stopper_Min_Back_Up AND Inputs.RC_Tray_Stopper_Max_Back_Up AND ((NOT DON_LC_Con_Free_Back AND NOT Settings.Option_InductiveTraydetection) OR ((NOT DON_IS_Con_In_Pos_Back OR NOT DON_IS_Con_In_Pos_Front) AND Settings.Option_InductiveTraydetection)) AND (DatAControl.OUT.Warning04 = WORD#0)) OR NOT Cyc_LoadBench.Step00 OR MachineMode.Manual;
(* Rung 104: Chain conveyer desired forward in automatic *)
ChainDesiredFWD_Auto := (Cyc_LoadBench.Step01 AND NOT Cyc_LoadBench.Step03 AND Cyc_LoadBench.Back) OR (Cyc_UnloadBench.Step01 AND NOT Cyc_UnloadBench.Step03 AND Cyc_UnloadBench.Front AND FrontCommIn.RequestSignal);
(* Rung 105: Chain conveyer desired backward in automatic *)
ChainDesiredREV_Auto := (Cyc_LoadBench.Step01 AND NOT Cyc_LoadBench.Step03 AND Cyc_LoadBench.Front) OR (Cyc_UnloadBench.Step01 AND NOT Cyc_UnloadBench.Step03 AND Cyc_UnloadBench.Back AND BackCommIn.RequestSignal);
(* Rung 106: Chain conveyer desired forward/ backward in manual *)
ManualControl_Chain(Enable := Enable, I_ManualMode := MachineMode.Manual, I_ManualOut := Commands.Chain.Out, I_ManualIn := Commands.Chain.In, I_ManualStop := Commands.Chain.Stop, O_ManualIn => ChainDesiredREV_Manual, O_ManualOut => ChainDesiredFWD_Manual);

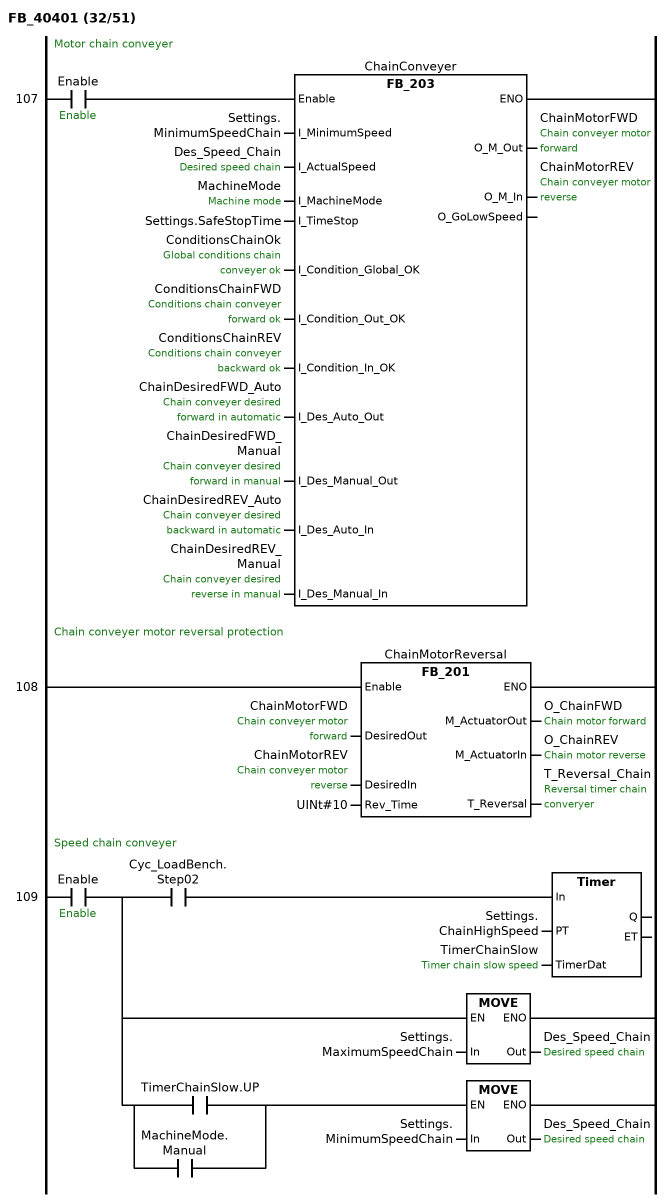
(* Rung 107: Motor chain conveyer *)
ChainConveyer(Enable := Enable, I_MinimumSpeed := Settings.MinimumSpeedChain, I_ActualSpeed := Des_Speed_Chain, I_MachineMode := MachineMode, I_TimeStop := Settings.SafeStopTime, I_Condition_Global_OK := ConditionsChainOk, I_Condition_Out_OK := ConditionsChainFWD, I_Condition_In_OK := ConditionsChainREV, I_Des_Auto_Out := ChainDesiredFWD_Auto, I_Des_Manual_Out := ChainDesiredFWD_Manual, I_Des_Auto_In := ChainDesiredREV_Auto, I_Des_Manual_In := ChainDesiredREV_Manual, O_M_Out => ChainMotorFWD, O_M_In => ChainMotorREV);
(* Rung 108: Chain conveyer motor reversal protection *)
ChainMotorReversal(Enable := TRUE, DesiredOut := ChainMotorFWD, DesiredIn := ChainMotorREV, Rev_Time := UINt#10, M_ActuatorOut => O_ChainFWD, M_ActuatorIn => O_ChainREV, T_Reversal => T_Reversal_Chain);
(* Rung 109: Speed chain conveyer *)
_t56 := Timer(In := Enable AND Cyc_LoadBench.Step02, PT := Settings.ChainHighSpeed, TimerDat := TimerChainSlow);
IF Enable THEN Des_Speed_Chain := Settings.MaximumSpeedChain; END_IF;
IF Enable AND (TimerChainSlow.UP OR MachineMode.Manual) THEN
    Des_Speed_Chain := Settings.MinimumSpeedChain;
END_IF;

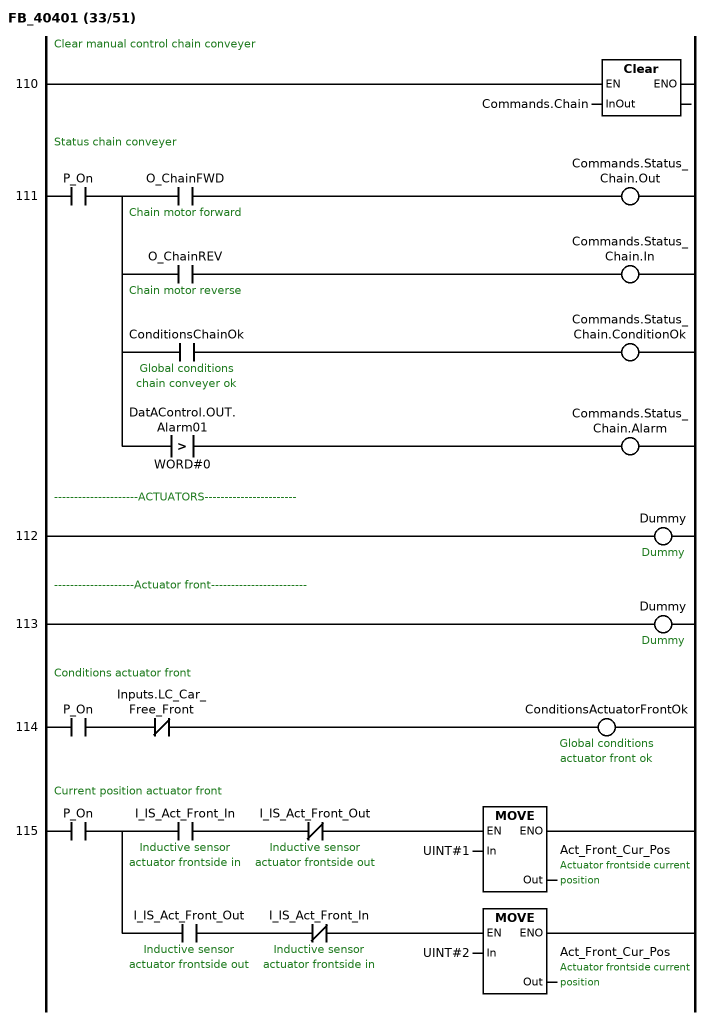
(* Rung 110: Clear manual control chain conveyer *)
Clear(InOut := Commands.Chain);
(* Rung 111: Status chain conveyer *)
Commands.Status_Chain.Out := P_On AND O_ChainFWD;
Commands.Status_Chain.In := P_On AND O_ChainREV;
Commands.Status_Chain.ConditionOk := P_On AND ConditionsChainOk;
Commands.Status_Chain.Alarm := P_On AND (DatAControl.OUT.Alarm01 > WORD#0);
(* Rung 112: ---------------------ACTUATORS----------------------- *)
Dummy := TRUE;
(* Rung 113: --------------------Actuator front------------------------ *)
Dummy := TRUE;
(* Rung 114: Conditions actuator front *)
ConditionsActuatorFrontOk := P_On AND NOT Inputs.LC_Car_Free_Front;
(* Rung 115: Current position actuator front *)
IF P_On AND I_IS_Act_Front_In AND NOT I_IS_Act_Front_Out THEN Act_Front_Cur_Pos := UINT#1; END_IF;
IF P_On AND I_IS_Act_Front_Out AND NOT I_IS_Act_Front_In THEN Act_Front_Cur_Pos := UINT#2; END_IF;

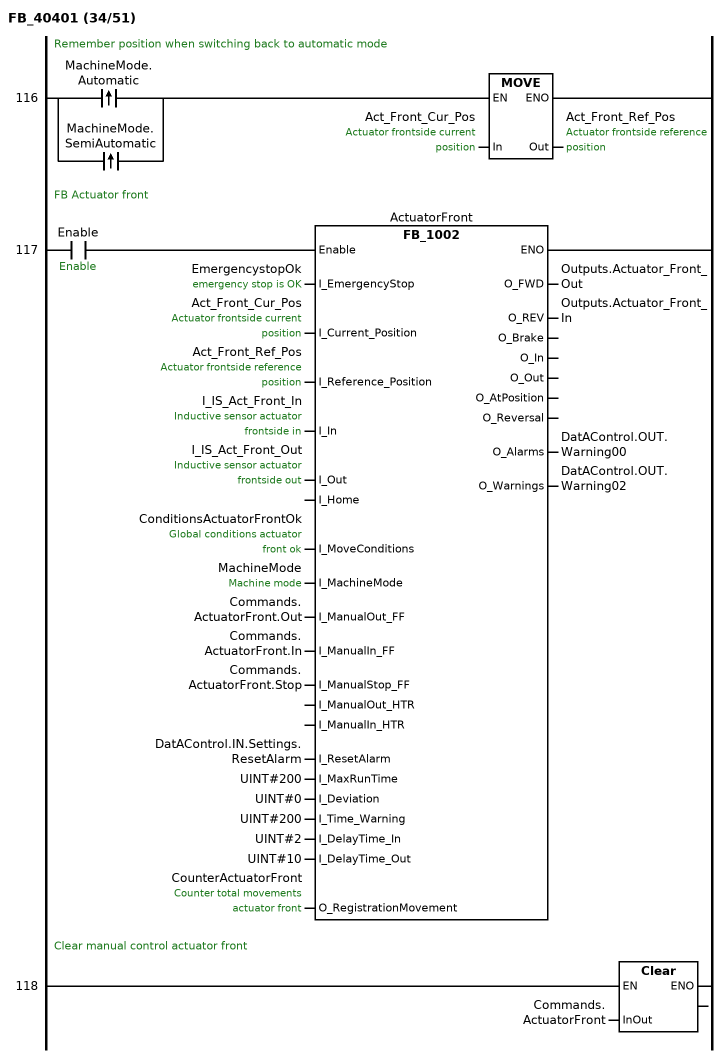
(* Rung 116: Remember position when switching back to automatic mode *)
_e57(CLK := MachineMode.Automatic);
_e58(CLK := MachineMode.SemiAutomatic);
IF _e57.Q OR _e58.Q THEN Act_Front_Ref_Pos := Act_Front_Cur_Pos; END_IF;
(* Rung 117: FB Actuator front *)
ActuatorFront(Enable := Enable, I_EmergencyStop := EmergencystopOk, I_Current_Position := Act_Front_Cur_Pos, I_Reference_Position := Act_Front_Ref_Pos, I_In := I_IS_Act_Front_In, I_Out := I_IS_Act_Front_Out, I_MoveConditions := ConditionsActuatorFrontOk, I_MachineMode := MachineMode, I_ManualOut_FF := Commands.ActuatorFront.Out, I_ManualIn_FF := Commands.ActuatorFront.In, I_ManualStop_FF := Commands.ActuatorFront.Stop, I_ResetAlarm := DatAControl.IN.Settings.ResetAlarm, I_MaxRunTime := UINT#200, I_Deviation := UINT#0, I_Time_Warning := UINT#200, I_DelayTime_In := UINT#2, I_DelayTime_Out := UINT#10, O_RegistrationMovement := CounterActuatorFront, O_FWD => Outputs.Actuator_Front_Out, O_REV => Outputs.Actuator_Front_In, O_Alarms => DatAControl.OUT.Warning00, O_Warnings => DatAControl.OUT.Warning02);
(* Rung 118: Clear manual control actuator front *)
Clear(InOut := Commands.ActuatorFront);

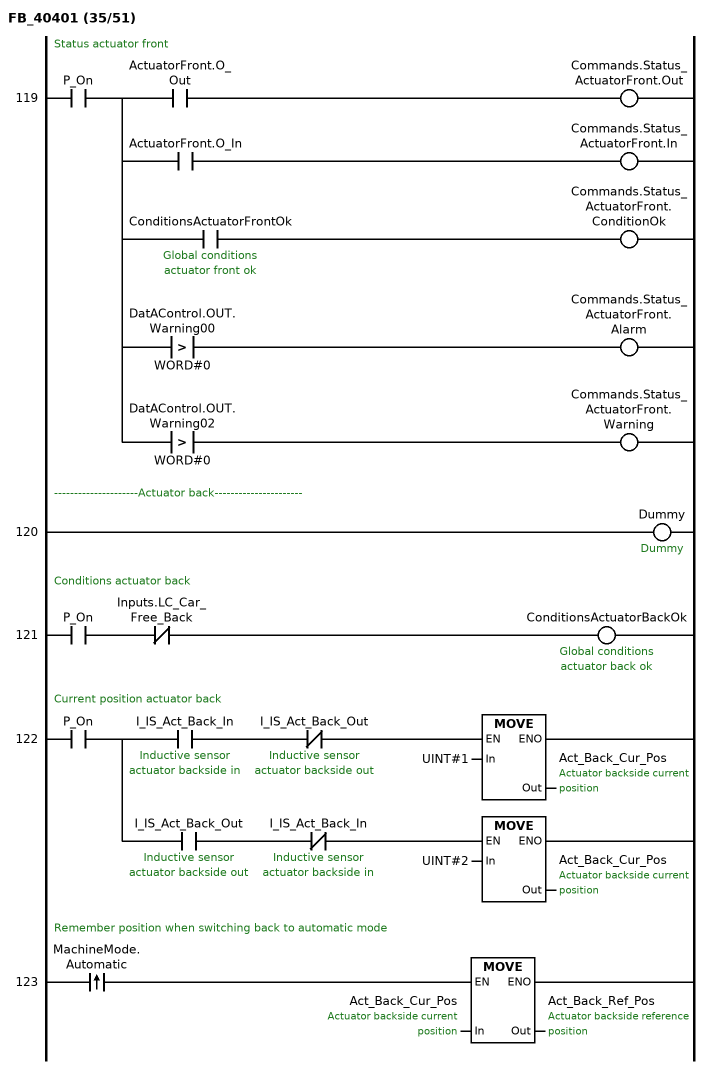
(* Rung 119: Status actuator front *)
Commands.Status_ActuatorFront.Out := P_On AND ActuatorFront.O_Out;
Commands.Status_ActuatorFront.In := P_On AND ActuatorFront.O_In;
Commands.Status_ActuatorFront.ConditionOk := P_On AND ConditionsActuatorFrontOk;
Commands.Status_ActuatorFront.Alarm := P_On AND (DatAControl.OUT.Warning00 > WORD#0);
Commands.Status_ActuatorFront.Warning := P_On AND (DatAControl.OUT.Warning02 > WORD#0);
(* Rung 120: ---------------------Actuator back---------------------- *)
Dummy := TRUE;
(* Rung 121: Conditions actuator back *)
ConditionsActuatorBackOk := P_On AND NOT Inputs.LC_Car_Free_Back;
(* Rung 122: Current position actuator back *)
IF P_On AND I_IS_Act_Back_In AND NOT I_IS_Act_Back_Out THEN Act_Back_Cur_Pos := UINT#1; END_IF;
IF P_On AND I_IS_Act_Back_Out AND NOT I_IS_Act_Back_In THEN Act_Back_Cur_Pos := UINT#2; END_IF;
(* Rung 123: Remember position when switching back to automatic mode *)
_e59(CLK := MachineMode.Automatic);
IF _e59.Q THEN Act_Back_Ref_Pos := Act_Back_Cur_Pos; END_IF;

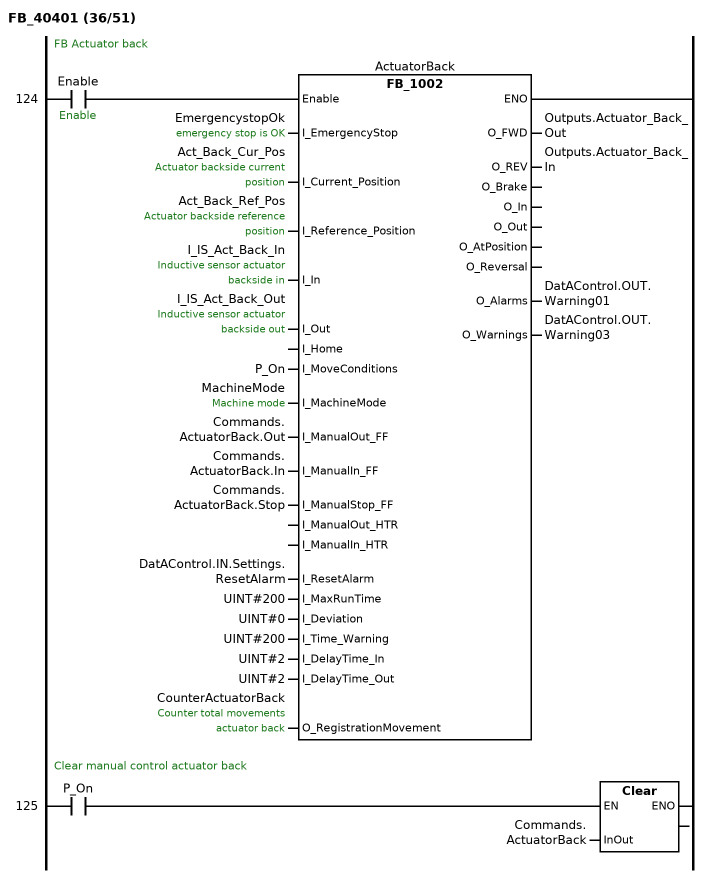
(* Rung 124: FB Actuator back *)
ActuatorBack(Enable := Enable, I_EmergencyStop := EmergencystopOk, I_Current_Position := Act_Back_Cur_Pos, I_Reference_Position := Act_Back_Ref_Pos, I_In := I_IS_Act_Back_In, I_Out := I_IS_Act_Back_Out, I_MoveConditions := P_On, I_MachineMode := MachineMode, I_ManualOut_FF := Commands.ActuatorBack.Out, I_ManualIn_FF := Commands.ActuatorBack.In, I_ManualStop_FF := Commands.ActuatorBack.Stop, I_ResetAlarm := DatAControl.IN.Settings.ResetAlarm, I_MaxRunTime := UINT#200, I_Deviation := UINT#0, I_Time_Warning := UINT#200, I_DelayTime_In := UINT#2, I_DelayTime_Out := UINT#2, O_RegistrationMovement := CounterActuatorBack, O_FWD => Outputs.Actuator_Back_Out, O_REV => Outputs.Actuator_Back_In, O_Alarms => DatAControl.OUT.Warning01, O_Warnings => DatAControl.OUT.Warning03);
(* Rung 125: Clear manual control actuator back *)
IF P_On THEN Clear(InOut := Commands.ActuatorBack); END_IF;

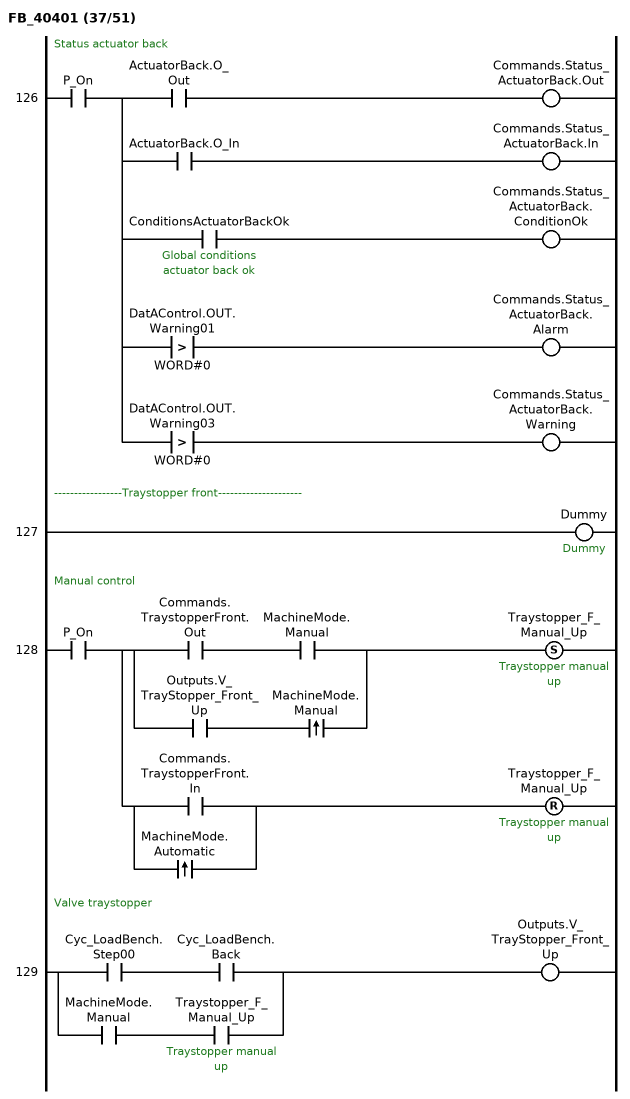
(* Rung 126: Status actuator back *)
Commands.Status_ActuatorBack.Out := P_On AND ActuatorBack.O_Out;
Commands.Status_ActuatorBack.In := P_On AND ActuatorBack.O_In;
Commands.Status_ActuatorBack.ConditionOk := P_On AND ConditionsActuatorBackOk;
Commands.Status_ActuatorBack.Alarm := P_On AND (DatAControl.OUT.Warning01 > WORD#0);
Commands.Status_ActuatorBack.Warning := P_On AND (DatAControl.OUT.Warning03 > WORD#0);
(* Rung 127: -----------------Traystopper front--------------------- *)
Dummy := TRUE;
(* Rung 128: Manual control *)
_e60(CLK := MachineMode.Manual);
IF P_On AND ((Commands.TraystopperFront.Out AND MachineMode.Manual) OR (Outputs.V_TrayStopper_Front_Up AND _e60.Q)) THEN
    Traystopper_F_Manual_Up := TRUE;
END_IF;
_e61(CLK := MachineMode.Automatic);
IF P_On AND (Commands.TraystopperFront.In OR _e61.Q) THEN Traystopper_F_Manual_Up := FALSE; END_IF;
(* Rung 129: Valve traystopper *)
Outputs.V_TrayStopper_Front_Up := (Cyc_LoadBench.Step00 AND Cyc_LoadBench.Back) OR (MachineMode.Manual AND Traystopper_F_Manual_Up);

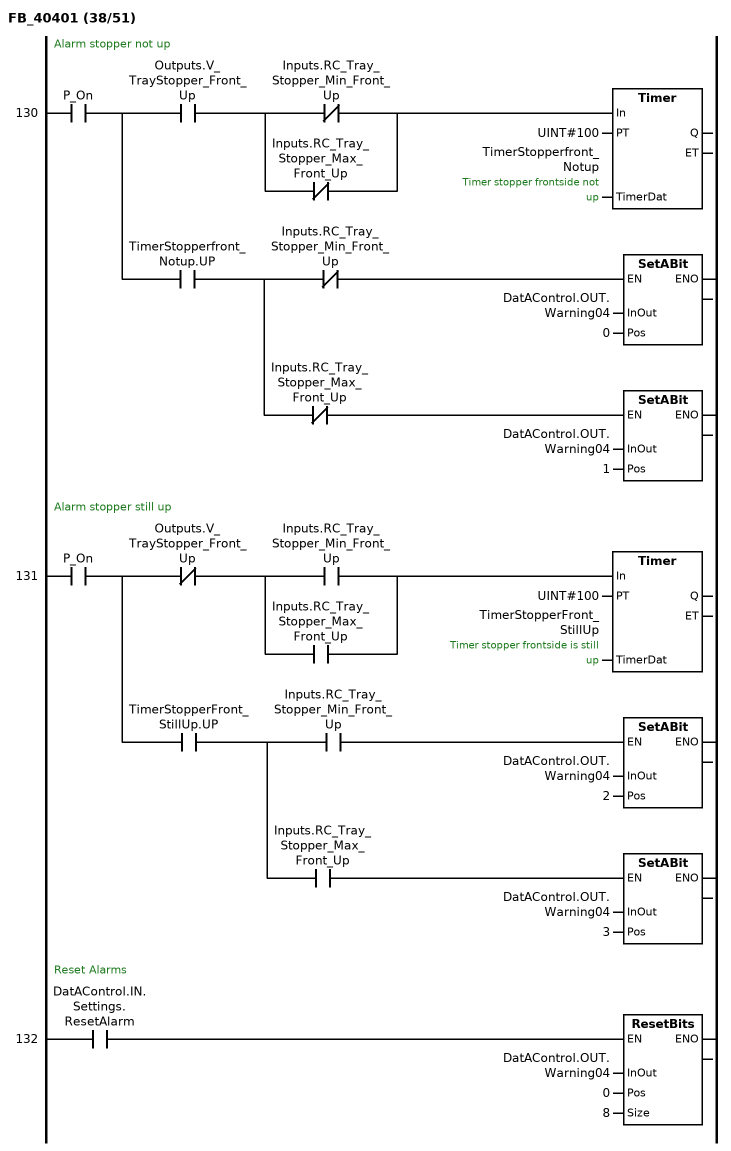
(* Rung 130: Alarm stopper not up *)
_t62 := Timer(In := P_On AND Outputs.V_TrayStopper_Front_Up AND (NOT Inputs.RC_Tray_Stopper_Min_Front_Up OR NOT Inputs.RC_Tray_Stopper_Max_Front_Up), PT := UINT#100, TimerDat := TimerStopperfront_Notup);
IF P_On AND TimerStopperfront_Notup.UP AND NOT Inputs.RC_Tray_Stopper_Min_Front_Up THEN
    SetABit(InOut := DatAControl.OUT.Warning04, Pos := 0);
END_IF;
IF P_On AND TimerStopperfront_Notup.UP AND NOT Inputs.RC_Tray_Stopper_Max_Front_Up THEN
    SetABit(InOut := DatAControl.OUT.Warning04, Pos := 1);
END_IF;
(* Rung 131: Alarm stopper still up *)
_t63 := Timer(In := P_On AND NOT Outputs.V_TrayStopper_Front_Up AND (Inputs.RC_Tray_Stopper_Min_Front_Up OR Inputs.RC_Tray_Stopper_Max_Front_Up), PT := UINT#100, TimerDat := TimerStopperFront_StillUp);
IF P_On AND TimerStopperFront_StillUp.UP AND Inputs.RC_Tray_Stopper_Min_Front_Up THEN
    SetABit(InOut := DatAControl.OUT.Warning04, Pos := 2);
END_IF;
IF P_On AND TimerStopperFront_StillUp.UP AND Inputs.RC_Tray_Stopper_Max_Front_Up THEN
    SetABit(InOut := DatAControl.OUT.Warning04, Pos := 3);
END_IF;
(* Rung 132: Reset Alarms *)
IF DatAControl.IN.Settings.ResetAlarm THEN
    ResetBits(InOut := DatAControl.OUT.Warning04, Pos := 0, Size := 8);
END_IF;

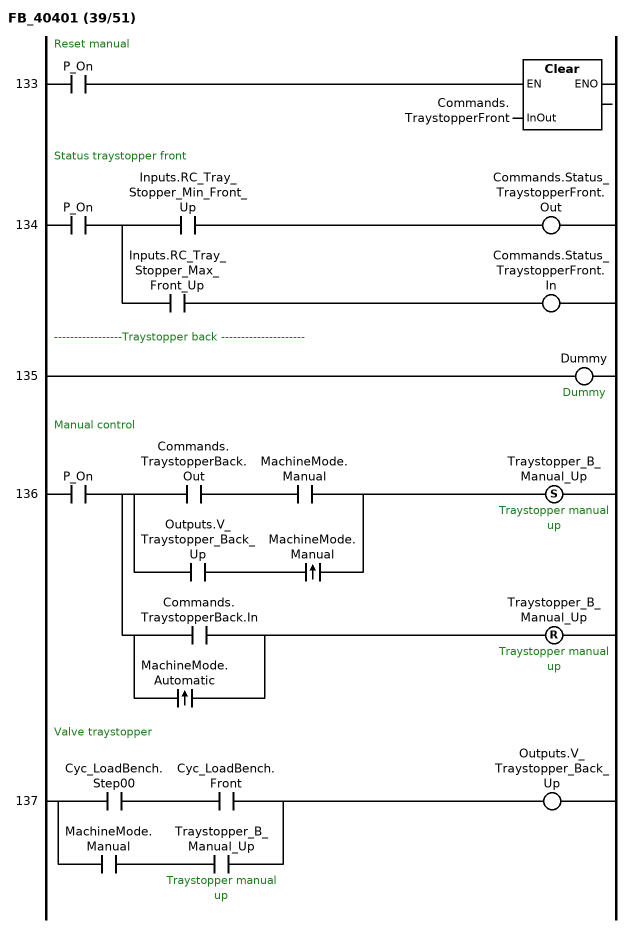
(* Rung 133: Reset manual *)
IF P_On THEN Clear(InOut := Commands.TraystopperFront); END_IF;
(* Rung 134: Status traystopper front *)
Commands.Status_TraystopperFront.Out := P_On AND Inputs.RC_Tray_Stopper_Min_Front_Up;
Commands.Status_TraystopperFront.In := P_On AND Inputs.RC_Tray_Stopper_Max_Front_Up;
(* Rung 135: -----------------Traystopper back --------------------- *)
Dummy := TRUE;
(* Rung 136: Manual control *)
_e64(CLK := MachineMode.Manual);
IF P_On AND ((Commands.TraystopperBack.Out AND MachineMode.Manual) OR (Outputs.V_Traystopper_Back_Up AND _e64.Q)) THEN
    Traystopper_B_Manual_Up := TRUE;
END_IF;
_e65(CLK := MachineMode.Automatic);
IF P_On AND (Commands.TraystopperBack.In OR _e65.Q) THEN Traystopper_B_Manual_Up := FALSE; END_IF;
(* Rung 137: Valve traystopper *)
Outputs.V_Traystopper_Back_Up := (Cyc_LoadBench.Step00 AND Cyc_LoadBench.Front) OR (MachineMode.Manual AND Traystopper_B_Manual_Up);

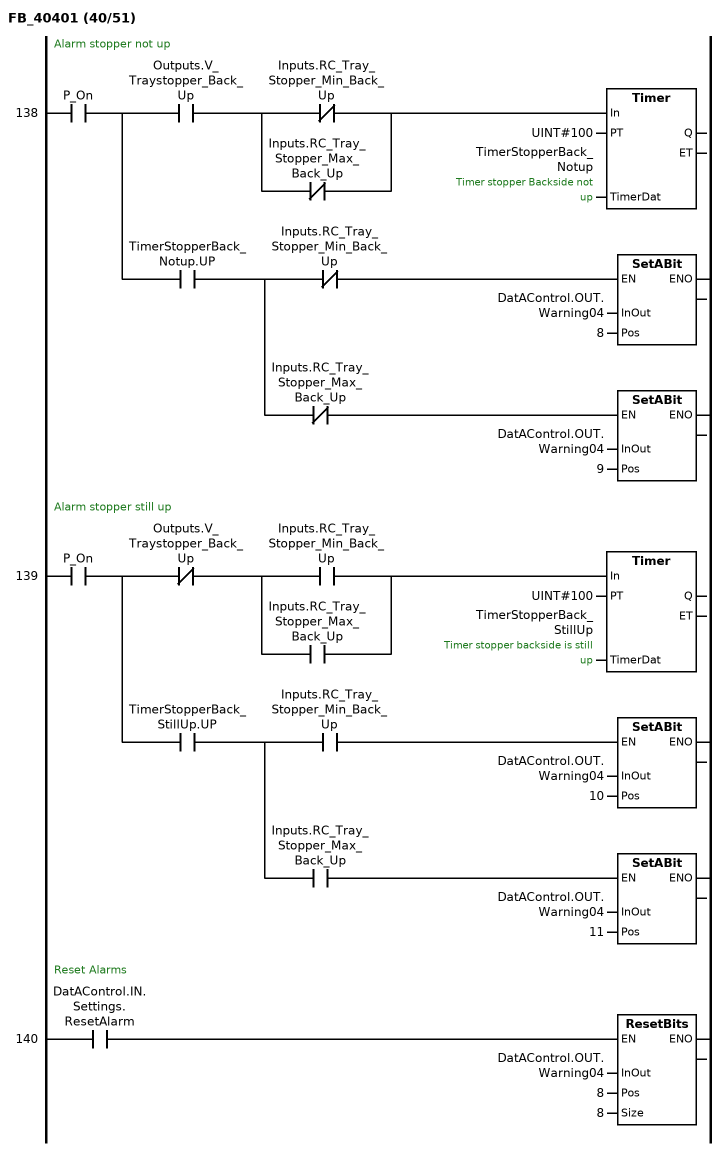
(* Rung 138: Alarm stopper not up *)
_t66 := Timer(In := P_On AND Outputs.V_Traystopper_Back_Up AND (NOT Inputs.RC_Tray_Stopper_Min_Back_Up OR NOT Inputs.RC_Tray_Stopper_Max_Back_Up), PT := UINT#100, TimerDat := TimerStopperBack_Notup);
IF P_On AND TimerStopperBack_Notup.UP AND NOT Inputs.RC_Tray_Stopper_Min_Back_Up THEN
    SetABit(InOut := DatAControl.OUT.Warning04, Pos := 8);
END_IF;
IF P_On AND TimerStopperBack_Notup.UP AND NOT Inputs.RC_Tray_Stopper_Max_Back_Up THEN
    SetABit(InOut := DatAControl.OUT.Warning04, Pos := 9);
END_IF;
(* Rung 139: Alarm stopper still up *)
_t67 := Timer(In := P_On AND NOT Outputs.V_Traystopper_Back_Up AND (Inputs.RC_Tray_Stopper_Min_Back_Up OR Inputs.RC_Tray_Stopper_Max_Back_Up), PT := UINT#100, TimerDat := TimerStopperBack_StillUp);
IF P_On AND TimerStopperBack_StillUp.UP AND Inputs.RC_Tray_Stopper_Min_Back_Up THEN
    SetABit(InOut := DatAControl.OUT.Warning04, Pos := 10);
END_IF;
IF P_On AND TimerStopperBack_StillUp.UP AND Inputs.RC_Tray_Stopper_Max_Back_Up THEN
    SetABit(InOut := DatAControl.OUT.Warning04, Pos := 11);
END_IF;
(* Rung 140: Reset Alarms *)
IF DatAControl.IN.Settings.ResetAlarm THEN
    ResetBits(InOut := DatAControl.OUT.Warning04, Pos := 8, Size := 8);
END_IF;

